(* Logix 5000 project; controller CLASE_1 Emulate 5570 rev 28.11; software revision 28.02 *)

TASK MainTask (continuous, watchdog 500 ms) : MainProgram
TASK TASK_A (periodic, rate 50 ms, priority 5, watchdog 150 ms) : Equipos_TK_100, Equipos_TK_200, Equipos_TK_300
TASK Task_B_100ms_Secuencias (periodic, rate 100 ms, priority 6, watchdog 300 ms) : SEC_Proceso_Chocolate_SFC
TASK Task_C_200ms (periodic, rate 200 ms, priority 7, watchdog 600 ms) : PID_Controllers

MODULES
   Local : Emulate 5570 (ICP 9, rev 28.11)
      Input_Digital_1 : 1756-IA16 (ICP 5, rev 3.1, Input RPI 20 ms)
      Output_Digital_2 : vendor 1 type 7 code 13 (ICP 6, rev 3.1, Output RPI 20 ms)
      input_analogica_1 : 1756-IF16 (ICP 7, rev 1.1, Input RPI 100 ms)
      Output_analogico_2 : 1756-OF8 (ICP 4, rev 1.1, Output RPI 12 ms)
END_MODULES

TYPE P_DescList :   // Code / Description List Entry
STRUCT
   Code : DINT;   // Code for which to look up Description
   Desc : STRING_40;   // Description for given Code
END_STRUCT
END_TYPE

TYPE STRING_12 :
STRUCT
   LEN : DINT;
   DATA : SINT[12];
END_STRUCT
END_TYPE

TYPE STRING_16 :
STRUCT
   LEN : DINT;
   DATA : SINT[16];
END_STRUCT
END_TYPE

TYPE STRING_20 :
STRUCT
   LEN : DINT;
   DATA : SINT[20];
END_STRUCT
END_TYPE

TYPE STRING_40 :
STRUCT
   LEN : DINT;
   DATA : SINT[40];
END_STRUCT
END_TYPE

TYPE STRING_8 :
STRUCT
   LEN : DINT;
   DATA : SINT[8];
END_STRUCT
END_TYPE

TYPE STRING_NavTag :   // Navigation Tag
STRUCT
   LEN : DINT;
   DATA : SINT[20];
END_STRUCT
END_TYPE

ADD_ON_INSTRUCTION P_AIn   (* revision 3.5 02 Release, vendor Rockwell Automation, ExecutePrescan, ExecuteEnableInFalse *)
// Analog Input
// Revision note:
// See V3.5-xx Release Notes for details. Added Cfg_UseChanSrcQ to make SrcQ use independent of Cfg_HasChanObj, which is for navigation only.
// Help:
// Copyright © Rockwell Automation, Inc.  All Rights Reserved.
// This Instruction monitors an Analog Input from a flow, level, pressure,
// temperature, or any other analog sensor, and provides:
// *  Scaling, from Input (Raw) to PV (Engineering) Units
// *  High-High, High, Low and Low-Low Status and Alarms, with Gate
// inputs and configurable on-delay, off-delay and gate delay times
// *  Monitoring of bad/uncertain PV status, floating point exceptions
// and out-of-range conditions, with PV Fail alarm
// *  Setting of a simulated input signal for process simulation
// *  Capturing of the lowest and highest PV excursion values
// *  Program and Operator Settings for Status Thresholds
// *  Configurable threshold deadbands and out of range limits
// *  Maintenance Commands to allow manual override of the input signal (Substitute PV)
// Modes are provided by a P_Mode AOI instance.
// Alarms are provided by P_Alarm AOI instances.
// Status gating provided by P_Gate AOI instances.
// Modes of operation: Operator, Program, Maintenance
VAR_INPUT
   Inp_PV : REAL; {visible}   // Input Signal (process variable) from Sensor
   Inp_PVSrcQ : SINT;   // Input Source and Quality (from Channel object, if available) (enum)
   Inp_PVBad : BOOL;   // 1=PV or I/O Comms Status Bad, 0=OK
   Inp_PVUncertain : BOOL;   // 1=PV Value Not Reliable, 0=OK
   Inp_Sim : BOOL;   // 1=Use simulated PV (Set_SimPV); 0=Use Input (Inp_PV)
   Inp_HiHiGate : ALIAS FOR HiHiGate.Inp_Gate;   // High-High Status Gate, 1=enabled
   Inp_HiGate : ALIAS FOR HiGate.Inp_Gate;   // High Status Gate, 1=enabled
   Inp_LoGate : ALIAS FOR LoGate.Inp_Gate;   // Low Status Gate, 1=enabled
   Inp_LoLoGate : ALIAS FOR LoLoGate.Inp_Gate;   // Low-Low Status Gate, 1=enabled
   Inp_FailGate : ALIAS FOR FailGate.Inp_Gate;   // Fail Status Gate, 1=enabled
   Inp_Reset : BOOL;   // 1=Reset all Alarms requiring reset
   Cfg_NoSubstPV : BOOL;   // 1=Disallow selection of Substitute PV
   Cfg_SetTrack : BOOL := 1;   // 1=PSets track OSets in Oper, OSets track PSets in Prog, 0=no tracking
   Cfg_HasChanObj : BOOL;   // 1=Tells HMI a Channel object (AIChan, etc.) is used for Inp_PV
   Cfg_UseChanSrcQ : BOOL;   // 1=Pass thru connected Channel's SrcQ value, 0=generate SrcQ
   Cfg_PCmdClear : ALIAS FOR Mode.Cfg_PCmdClear;
   Cfg_ProgDefault : ALIAS FOR Mode.Cfg_ProgDefault;
   Cfg_HasHiHiAlm : ALIAS FOR HiHi.Cfg_Exists;   // 1=High-High Alarm exists and will be checked
   Cfg_HasHiAlm : ALIAS FOR Hi.Cfg_Exists;   // 1=High Alarm exists and will be checked
   Cfg_HasLoAlm : ALIAS FOR Lo.Cfg_Exists;   // 1=Low Alarm exists and will be checked
   Cfg_HasLoLoAlm : ALIAS FOR LoLo.Cfg_Exists;   // 1=Low-Low Alarm exists and will be checked
   Cfg_HasFailAlm : ALIAS FOR Fail.Cfg_Exists;   // 1=Analog Input Failure Alarm exists and will be checked
   Cfg_HiHiResetReqd : ALIAS FOR HiHi.Cfg_ResetReqd;   // 1=Reset required to clear High-High Alarm
   Cfg_HiResetReqd : ALIAS FOR Hi.Cfg_ResetReqd;   // 1=Reset required to clear High Alarm
   Cfg_LoResetReqd : ALIAS FOR Lo.Cfg_ResetReqd;   // 1=Reset required to clear Low Alarm
   Cfg_LoLoResetReqd : ALIAS FOR LoLo.Cfg_ResetReqd;   // 1=Reset required to clear Low-Low Alarm
   Cfg_FailResetReqd : ALIAS FOR Fail.Cfg_ResetReqd;   // 1=Reset required to clear Analog InputFailure Alarm
   Cfg_HiHiAckReqd : ALIAS FOR HiHi.Cfg_AckReqd;   // 1=Acknowledge required for High-High Alarm
   Cfg_HiAckReqd : ALIAS FOR Hi.Cfg_AckReqd;   // 1=Acknowledge required for High Alarm
   Cfg_LoAckReqd : ALIAS FOR Lo.Cfg_AckReqd;   // 1=Acknlowledge required for Low Alarm
   Cfg_LoLoAckReqd : ALIAS FOR LoLo.Cfg_AckReqd;   // 1=Acknowledge required for Low-Low Alarm
   Cfg_FailAckReqd : ALIAS FOR Fail.Cfg_AckReqd;   // 1=Acknowledge required for Analog Input Failure Alarm
   Cfg_HiHiSeverity : ALIAS FOR HiHi.Cfg_Severity;   // High-High Alarm Severity: 1..250=Low, 251..500=Medium, 501..750=High, 751..1000=Urgent
   Cfg_HiSeverity : ALIAS FOR Hi.Cfg_Severity;   // High Alarm Severity: 1..250=Low, 251..500=Medium, 501..750=High, 751..1000=Urgent
   Cfg_LoSeverity : ALIAS FOR Lo.Cfg_Severity;   // Low Alarm Severity: 1..250=Low, 251..500=Medium, 501..750=High, 751..1000=Urgent
   Cfg_LoLoSeverity : ALIAS FOR LoLo.Cfg_Severity;   // Low-Low Alarm Severity: 1..250=Low, 251..500=Medium, 501..750=High, 751..1000=Urgent
   Cfg_FailSeverity : ALIAS FOR Fail.Cfg_Severity;   // Failure Alarm Severity: 1..250=Low, 251..500=Medium, 501..750=High, 751..1000=Urgent
   Cfg_InpRawMin : REAL;   // Input (unscaled) Minimum for Scaling
   Cfg_InpRawMax : REAL := 100.0;   // Input (unscaled) Maximum for Scaling
   Cfg_PVEUMin : REAL;   // PV (Output) Minimum for Scaling to EU
   Cfg_PVEUMax : REAL := 100.0;   // PV (Output) Maximum for Scaling to EU
   Cfg_FiltTC : REAL;   // PV Filter Time Constant (s), 0.0 = unfiltered
   Cfg_HiHiDB : REAL := 1.0;   // High-High Status Deadband (EU)
   Cfg_HiHiOnDly : ALIAS FOR HiHiGate.Cfg_OnDly;   // Minimum time above High-High Limit to raise Status (s)
   Cfg_HiHiOffDly : ALIAS FOR HiHiGate.Cfg_OffDly;   // Minimum time below High-High Limit (minus deadband) to clear Status (s)
   Cfg_HiHiGateDly : ALIAS FOR HiHiGate.Cfg_GateDly;   // High-High Status Gate Delay (s)
   Cfg_HiDB : REAL := 1.0;   // High Status Deadband (EU)
   Cfg_HiOnDly : ALIAS FOR HiGate.Cfg_OnDly;   // Minimum time above High Limit to raise Status (s)
   Cfg_HiOffDly : ALIAS FOR HiGate.Cfg_OffDly;   // Minimum time below High Limit (minus deadband) to clear Status (s)
   Cfg_HiGateDly : ALIAS FOR HiGate.Cfg_GateDly;   // High Status Gate Delay (s)
   Cfg_LoDB : REAL := 1.0;   // Low Status Deadband (EU)
   Cfg_LoOnDly : ALIAS FOR LoGate.Cfg_OnDly;   // Minimum time below Low Limit to raise Status (s)
   Cfg_LoOffDly : ALIAS FOR LoGate.Cfg_OffDly;   // Minimum time above Low Limit (plus deadband) to clear Status (s)
   Cfg_LoGateDly : ALIAS FOR LoGate.Cfg_GateDly;   // Low Status Gate Delay (s)
   Cfg_LoLoDB : REAL := 1.0;   // Low-Low Status Deadband (EU)
   Cfg_LoLoOnDly : ALIAS FOR LoLoGate.Cfg_OnDly;   // Minimum time below Low-Low Limit to raise Status (s)
   Cfg_LoLoOffDly : ALIAS FOR LoLoGate.Cfg_OffDly;   // Minimum time above Low-Low Limit (plus deadband) to clear Status (s)
   Cfg_LoLoGateDly : ALIAS FOR LoLoGate.Cfg_GateDly;   // Low-Low Status Gate Delay (s)
   Cfg_FailHiLim : REAL := 103.958336;   // Out-of-Range (fail) High Limit (EU)
   Cfg_FailLoLim : REAL := -2.0833333;   // Out-of-Range (fail) Low Limit (EU)
   Cfg_FailDB : REAL := 0.41666666;   // Out-of-Range (fail) High/Low Deadband (EU)
   Cfg_FailOnDly : ALIAS FOR FailGate.Cfg_OnDly;   // Minimum time Bad or Out of Range to raise Fail Status (s)
   Cfg_FailOffDly : ALIAS FOR FailGate.Cfg_OffDly;   // Minimum time OK or In Range to clear Fail Status (s)
   Cfg_FailGateDly : ALIAS FOR FailGate.Cfg_GateDly;   // Fail Status Gate Delay (s)
   PSet_Owner : DINT;   // Program Owner Request ID (non-zero) or Release (zero)
   PSet_HiHiLim : REAL := 1.5e+38;   // Program-Entered High-High Status Threshold (EU)
   PSet_HiLim : REAL := 1.5e+38;   // Program-Entered High Status Threshold (EU)
   PSet_LoLim : REAL := -1.5e+38;   // Program-Entered Low Status Threshold (EU)
   PSet_LoLoLim : REAL := -1.5e+38;   // Program-Entered Low-Low Status Threshold (EU)
   MSet_SubstPV : REAL;   // Maintenance-Entered Substitute PV (EU)
   OSet_HiHiLim : REAL := 1.5e+38;   // Operator-Entered High-High Status Threshold (EU)
   OSet_HiLim : REAL := 1.5e+38;   // Operator-Entered High Status Threshold (EU)
   OSet_LoLim : REAL := -1.5e+38;   // Operator-Entered Low Status Threshold (EU)
   OSet_LoLoLim : REAL := -1.5e+38;   // Operator-Entered Low-Low Status Threshold (EU)
   Set_SimPV : REAL;   // PV used in Simulation (Inp_Sim=1) (EU)
   PCmd_ClearCapt : BOOL;   // Program Command to Clear the captured min / max PV excursion values
   PCmd_Acq : ALIAS FOR Mode.PCmd_Acq;
   PCmd_Rel : ALIAS FOR Mode.PCmd_Rel;
   PCmd_Lock : ALIAS FOR Mode.PCmd_Lock;
   PCmd_Unlock : ALIAS FOR Mode.PCmd_Unlock;
   PCmd_Reset : BOOL;   // Program Command to Reset all Alarms requiring Reset
   PCmd_HiHiAck : ALIAS FOR HiHi.PCmd_Ack;   // Program Command to Acknowledge High-High Alarm
   PCmd_HiHiSuppress : ALIAS FOR HiHi.PCmd_Suppress;   // Program Command to Suppress High-High Alarm
   PCmd_HiHiUnsuppress : ALIAS FOR HiHi.PCmd_Unsuppress;   // Program Command to Unsuppress High-High Alarm
   PCmd_HiHiUnshelve : ALIAS FOR HiHi.PCmd_Unshelve;   // Program Command to Unshelve High-High Alarm
   PCmd_HiAck : ALIAS FOR Hi.PCmd_Ack;   // Program Command to Acknowledge High Alarm
   PCmd_HiSuppress : ALIAS FOR Hi.PCmd_Suppress;   // Program Command to Suppress High Alarm
   PCmd_HiUnsuppress : ALIAS FOR Hi.PCmd_Unsuppress;   // Program Command to Unsuppress High Alarm
   PCmd_HiUnshelve : ALIAS FOR Hi.PCmd_Unshelve;   // Program Command to Unshelve High Alarm
   PCmd_LoAck : ALIAS FOR Lo.PCmd_Ack;   // Program Command to Acknowledge Low Alarm
   PCmd_LoSuppress : ALIAS FOR Lo.PCmd_Suppress;   // Program Command to Suppress Low Alarm
   PCmd_LoUnsuppress : ALIAS FOR Lo.PCmd_Unsuppress;   // Program Command to Unsuppress Low Alarm
   PCmd_LoUnshelve : ALIAS FOR Lo.PCmd_Unshelve;   // Program Command to Unshelve Low Alarm
   PCmd_LoLoAck : ALIAS FOR LoLo.PCmd_Ack;   // Program Command to Acknowledge Low-Low Alarm
   PCmd_LoLoSuppress : ALIAS FOR LoLo.PCmd_Suppress;   // Program Command to Suppress Low-Low Alarm
   PCmd_LoLoUnsuppress : ALIAS FOR LoLo.PCmd_Unsuppress;   // Program Command to Unsuppress Low-Low Alarm
   PCmd_LoLoUnshelve : ALIAS FOR LoLo.PCmd_Unshelve;   // Program Command to Unshelve Low-Low Alarm
   PCmd_FailAck : ALIAS FOR Fail.PCmd_Ack;   // Program Command to Acknowldege Analog Input Failure Alarm
   PCmd_FailSuppress : ALIAS FOR Fail.PCmd_Suppress;   // Program Command to Suppress Analog Input Failure Alarm
   PCmd_FailUnsuppress : ALIAS FOR Fail.PCmd_Unsuppress;   // Program Command to Unsuppress Analog Input Failure Alarm
   PCmd_FailUnshelve : ALIAS FOR Fail.PCmd_Unshelve;   // Program Command to Unshelve Analog Input Failure Alarm
   MCmd_SubstPV : BOOL;   // Maintenance Command to use Substitute PV (override input)
   MCmd_InpPV : BOOL;   // Maintenance Command to use Input PV (normal)
   OCmd_ClearCapt : BOOL;   // Operator Command to Clear the captured min / max PV excursion values
   MCmd_Acq : ALIAS FOR Mode.MCmd_Acq;
   MCmd_Rel : ALIAS FOR Mode.MCmd_Rel;
   OCmd_AcqLock : ALIAS FOR Mode.OCmd_AcqLock;
   OCmd_Unlock : ALIAS FOR Mode.OCmd_UnlockRel;
   OCmd_Reset : BOOL;   // Operator Command to Reset all Alarms requiring Reset
   OCmd_ResetAckAll : BOOL;   // Operator Command to Reset and Acknowledge all Alarms
END_VAR
VAR_OUTPUT
   Val : REAL; {access Read Only, visible}   // Analog Value (after Substitute PV, if used)
   Val_InpPV : REAL; {access Read Only, visible}   // Analog Input Value (actual, before Substitute PV selection)
   Val_PVMinCapt : REAL := 1.5e+38; {access Read Only}   // Captured PV Minimum (excursion) since last cleared
   Val_PVMaxCapt : REAL := -1.5e+38; {access Read Only}   // Captured PV Maximum (excursion) since last cleared
   Val_PVEUMin : REAL; {access Read Only}   // Minimum of scaled range = MIN (Cfg_PVEUMin, Cfg_PVEUMax)
   Val_PVEUMax : REAL := 100.0; {access Read Only}   // Maximum of scaled range = MAX (Cfg_PVEUMin, Cfg_PVEUMax)
   SrcQ_IO : SINT; {access Read Only}   // Source and Quality of primary I/O (enumeration)
   SrcQ : SINT; {access Read Only}   // Source and Quality of primary Val/Sts (enumeration)
   Val_Fault : SINT; {access Read Only}   // Device Fault Status 0=none, 20=Lo, 21=Hi, 24=LoLo, 25=HiHi, 32=Fail, 34=CfgErr
   Val_Mode : ALIAS FOR Mode.Val; {access Read Only}
   Val_Owner : DINT; {access Read Only}   // Current Object Owner ID (0=not owned)
   Val_Notify : SINT; {access Read Only}   // Current Alarm Level and Acknowledgement (enumeration)
   Val_HiHiLim : REAL := 1.5e+38; {access Read Only, visible}   // Current High-High Status Threshold
   Val_HiLim : REAL := 1.5e+38; {access Read Only, visible}   // Current High Status Threshold
   Val_LoLim : REAL := -1.5e+38; {access Read Only, visible}   // Current Low Status Threshold
   Val_LoLoLim : REAL := -1.5e+38; {access Read Only, visible}   // Current Low-Low Status Threshold
   Sts_SubstPV : BOOL; {access Read Only}   // 1=Using Substitute PV (Input being overridden)
   Sts_InpPV : BOOL := 1; {access Read Only}   // 1=Using Input PV (normal)
   Sts_PVBad : BOOL; {access Read Only}   // 1=PV Bad quality or Out of Range
   Sts_PVUncertain : BOOL; {access Read Only}   // 1=PV Value is Uncertain (quality)
   Sts_MaintByp : BOOL; {access Read Only}   // 1=A Maintenance Bypass is Active, display icon
   Sts_AlmInh : BOOL; {access Read Only}   // 1=An Alarm is Shelved, Disabled or Suppressed: display icon
   Sts_Err : BOOL; {access Read Only, visible}   // 1=Error in Config (see detail Err_ bits for reason), display icon
   Err_Raw : BOOL; {access Read Only}   // 1=Error in Config: Raw Input Scaling Min = Max
   Err_EU : BOOL; {access Read Only}   // 1=Error in Config: Scaled EU Min = Max
   Err_Timer : BOOL; {access Read Only}   // 1=Error in Config: On Delay, Off Delay, Gate Delay Time Invalid (use 0 to 2147483 s)
   Err_Filt : BOOL; {access Read Only}   // 1=Error in Config: PV filter params (RateTime, TC)
   Err_DB : BOOL; {access Read Only}   // 1=Error in Config: a Status Deadband is < 0.0
   Err_Alarm : BOOL; {access Read Only}   // 1=Error in Config: Alarm Min On Time, Shelf Time, Severity
   Sts_Maint : ALIAS FOR Mode.Sts_Maint; {access Read Only}
   Sts_Prog : ALIAS FOR Mode.Sts_Prog; {access Read Only}
   Sts_Oper : ALIAS FOR Mode.Sts_Oper; {access Read Only}
   Sts_ProgOperLock : ALIAS FOR Mode.Sts_ProgOperLock; {access Read Only}
   Sts_NoMode : ALIAS FOR Mode.Sts_NoMode; {access Read Only}
   Sts_MAcqRcvd : ALIAS FOR Mode.Sts_MAcqRcvd; {access Read Only}
   Sts_HiHiCmp : ALIAS FOR HiHiGate.Inp;   // PV High-High comparison result 1=High-High
   Sts_HiHiGate : ALIAS FOR HiHiGate.Sts_Gate; {access Read Only}   // PV High-High Gate Delay Status, 1=done
   Sts_HiHi : ALIAS FOR HiHi.Inp;   // 1=Analog Input is above High-High limit
   Alm_HiHi : ALIAS FOR HiHi.Alm;   // 1=Analog Input is in High-High Alarm
   Ack_HiHi : ALIAS FOR HiHi.Ack;   // 1=High-High Alarm has been acknowledged
   Sts_HiHiDisabled : ALIAS FOR HiHi.Disabled;   // 1=High-High Alarm has been Disabled by Maintenancy
   Sts_HiHiSuppressed : ALIAS FOR HiHi.Suppressed;   // 1=High-High Alarm has been Suppressed by Program
   Sts_HiHiShelved : ALIAS FOR HiHi.Shelved;   // 1=High-High Alarm has been Shelved by Operator
   Sts_HiCmp : ALIAS FOR HiGate.Inp;   // PV High comparison result 1=High
   Sts_HiGate : ALIAS FOR HiGate.Sts_Gate; {access Read Only}   // PV High Gate Delay Status, 1=done
   Sts_Hi : ALIAS FOR Hi.Inp;   // 1=Analog Input is above High limit
   Alm_Hi : ALIAS FOR Hi.Alm;   // 1=Analog Input is in High Alarm
   Ack_Hi : ALIAS FOR Hi.Ack;   // 1=High Alarm has been acknowledged
   Sts_HiDisabled : ALIAS FOR Hi.Disabled;   // 1=High Alarm has been Disabled by Maintenance
   Sts_HiSuppressed : ALIAS FOR Hi.Suppressed;   // 1=High Alarm has been Suppressed by Program
   Sts_HiShelved : ALIAS FOR Hi.Shelved;   // 1=High Alarm has been Shelved by Operator
   Sts_LoCmp : ALIAS FOR LoGate.Inp;   // PV Low comparison result 1=Low
   Sts_LoGate : ALIAS FOR LoGate.Sts_Gate; {access Read Only}   // PV Low Gate Delay Status, 1=done
   Sts_Lo : ALIAS FOR Lo.Inp;   // 1=Analog Input is below Low limit
   Alm_Lo : ALIAS FOR Lo.Alm;   // 1=Analog Input is in Low Alarm
   Ack_Lo : ALIAS FOR Lo.Ack;   // 1=Low Alarm has been acknowledged
   Sts_LoDisabled : ALIAS FOR Lo.Disabled;   // 1=Low Alarm has been Disabled by Maintenance
   Sts_LoSuppressed : ALIAS FOR Lo.Suppressed;   // 1=Low Alarm has been Suppressed by Program
   Sts_LoShelved : ALIAS FOR Lo.Shelved;   // 1=Low Alarm has been Shelved by Operator
   Sts_LoLoCmp : ALIAS FOR LoLoGate.Inp;   // PV Low-Low comparison result 1=Low-Low
   Sts_LoLoGate : ALIAS FOR LoLoGate.Sts_Gate; {access Read Only}   // PV Low-Low Gate Delay Status, 1=done
   Sts_LoLo : ALIAS FOR LoLo.Inp;   // 1=Analog Input is below Low-Low limit
   Alm_LoLo : ALIAS FOR LoLo.Alm;   // 1=Analog Input is in Low-Low Alarm
   Ack_LoLo : ALIAS FOR LoLo.Ack;   // 1=Low-Low Alarm has been acknowledged
   Sts_LoLoDisabled : ALIAS FOR LoLo.Disabled;   // 1=Low-Low Alarm has been Disabled by Maintenance
   Sts_LoLoSuppressed : ALIAS FOR LoLo.Suppressed;   // 1=Low-Low Alarm has been Suppressed by Program
   Sts_LoLoShelved : ALIAS FOR LoLo.Shelved;   // 1=Low-Low Alarm has been Shelved by Operator
   Sts_FailCmp : ALIAS FOR FailGate.Inp;   // PV Fail comparison result 1=Out of Range
   Sts_FailGate : ALIAS FOR FailGate.Sts_Gate; {access Read Only}   // PV Fail Gate Delay Status, 1=done
   Sts_Fail : ALIAS FOR Fail.Inp;   // 1=Analog Input is Out of Range or PV Bad
   Alm_Fail : ALIAS FOR Fail.Alm;   // 1=Analog Input Failure Alarm (PV Bad or Out of Range)
   Ack_Fail : ALIAS FOR Fail.Ack;   // 1=Analog Input Failure Alarm has been acknowledged
   Sts_FailDisabled : ALIAS FOR Fail.Disabled;   // 1=Analog input Failure Alarm has been Disabled by Maintenance
   Sts_FailSuppressed : ALIAS FOR Fail.Suppressed;   // 1=Analog Input Failure Alarm has been Suppressed by Program
   Sts_FailShelved : ALIAS FOR Fail.Shelved;   // 1=Analog Input Failure Alarm has been Shelved by Operator
   Rdy_SubstPV : BOOL; {access Read Only}   // 1=Ready for MCmd_SubstPV
   Rdy_InpPV : BOOL; {access Read Only}   // 1=Ready for MCmd_InpPV
   Rdy_Reset : BOOL; {access Read Only}   // 1=At least one Alarm requires Reset
   Rdy_ResetAckAll : BOOL; {access Read Only}   // 1=At least one Alarm requires Reset or Acknowledgement
   Rdy_OSet : BOOL; {access Read Only}   // 1=Ready to receive OSets (enables data entry fields)
   P_AIn : BOOL;   // Unique Parameter Name for auto - discovery
END_VAR
VAR
   LoLo : P_Alarm := (Cfg_AckReqd := 1, Cfg_AllowShelve := 1, Cfg_AllowDisable := 1, Cfg_PCmdClear := 1, Cfg_Severity := 750, Cfg_AlmMinOnT := 5, PCfg_AllowExist := 1, Ack := 1);   // Low-Low Alarm
   Lo : P_Alarm := (Cfg_AckReqd := 1, Cfg_AllowShelve := 1, Cfg_AllowDisable := 1, Cfg_PCmdClear := 1, Cfg_Severity := 500, Cfg_AlmMinOnT := 5, PCfg_AllowExist := 1, Ack := 1);   // Low Alarm
   Hi : P_Alarm := (Cfg_AckReqd := 1, Cfg_AllowShelve := 1, Cfg_AllowDisable := 1, Cfg_PCmdClear := 1, Cfg_Severity := 500, Cfg_AlmMinOnT := 5, PCfg_AllowExist := 1, Ack := 1);   // High Alarm
   HiHi : P_Alarm := (Cfg_AckReqd := 1, Cfg_AllowShelve := 1, Cfg_AllowDisable := 1, Cfg_PCmdClear := 1, Cfg_Severity := 750, Cfg_AlmMinOnT := 5, PCfg_AllowExist := 1, Ack := 1);   // High-High Alarm
   Mode : P_Mode := (Cfg_PCmdClear := 1, Cfg_OvrdOverLock := 1, Sts_Oper := 1, Rdy_MRel := 1, Rdy_OAcq := 1);   // Analog Input Mode Selection
   Cfg_EU : STRING_8 := '%';   // Engineering Units for display on HMI
   Cfg_Tag : STRING_20 := 'P_AIn';   // Tagname for display on HMI
   Cfg_Label : STRING_20 := 'Analog Input';   // Label for graphic symbol displayed on HMI
   Cfg_Desc : STRING_40 := 'Analog Input';   // Description for display on HMI
   Fail : P_Alarm := (Cfg_AckReqd := 1, Cfg_AllowShelve := 1, Cfg_AllowDisable := 1, Cfg_PCmdClear := 1, Cfg_Severity := 1000, Cfg_AlmMinOnT := 5, PCfg_AllowExist := 1, Ack := 1);   // Analog Input Failure Alarm (bad quality or out of range)
   Wrk_Notify : SINT; {access None}   // Buffer for building Val_Notify
   Inf_Tab : SINT;   // Tab to display (FTView ME)
   Wrk_Fault : SINT; {access None}   // Buffer for building Val_Fault
   Wrk_SrcQ : SINT; {access None}   // Register for building Source / Quality enumeration
   Wrk_SubstPV : BOOL; {access None}   // Internal flag: Using Substitute PV
   Wrk_UnfiltPV : REAL; {access None}   // Unfiltered PV, input to 1st order filter
   Wrk_Alpha : REAL; {access None}   // Filter multiplier = (1 / (1+TC/dT) )
   Wrk_ScanT : TIMER := (PRE := 2147483647); {access None}   // Scan Timer (milliseconds, always runs)
   Wrk_ScanTime : REAL; {access None}   // Time since this instance was last scanned
   Wrk_FiltPV : REAL; {access None}   // Filtered PV
   Wrk_ValidONS : BOOL; {access None}   // Selected PV goes from Infinite or Not a Number to VALID
   Wrk_SelPVDINT : DINT; {access None}   // Selected PV check for Infinite or Non A Number
   Wrk_SelPVInfNaN : BOOL; {access None}   // Selected PV (Input or Substitute) is Infinite or NaN
   Inf_Type : STRING_16 := 'P_AIn'; {access Read Only}   // Must contain AOI name, used for HMI and Information S/W
   Wrk_Fail : BOOL; {access None}   // Internal flag: Fail Status
   Wrk_LoLo : BOOL; {access None}   // Internal flag: Low-Low Status
   Wrk_Lo : BOOL; {access None}   // Internal flag: Low Status
   Wrk_Hi : BOOL; {access None}   // Internal flag: High Status
   Wrk_HiHi : BOOL; {access None}   // Internal flag: High-High Status
   FailGate : P_Gate := (Inp_Gate := 1);   // Fail Alarm Gate / Delay Block
   LoLoGate : P_Gate := (Inp_Gate := 1);   // Low-Low Alarm Gate / Delay Block
   LoGate : P_Gate := (Inp_Gate := 1);   // Low Alarm Gate / Delay Block
   HiHiGate : P_Gate := (Inp_Gate := 1);   // High-High Alarm Gate / Delay Block
   HiGate : P_Gate := (Inp_Gate := 1);   // High Alarm Gate / Delay Block
   Wrk_InpInfNaN : BOOL; {access None}   // Input is Infinite or Not a Number
   Wrk_InpDINT : DINT; {access None}   // Input REAL bit pattern as a DINT (check for Inf/NaN)
   Inf_Lib : STRING_12 := 'RA-BAS'; {access Read Only}   // Display Library for Faceplate call-up
   Wrk_InpFail : BOOL; {access None}   // Input Fail: out of range
END_VAR

ROUTINE EnableInFalse   (* ladder *)
// Off-Scan: no Val update or alarm checking.  PV Bad Quality ("stale") is asserted.
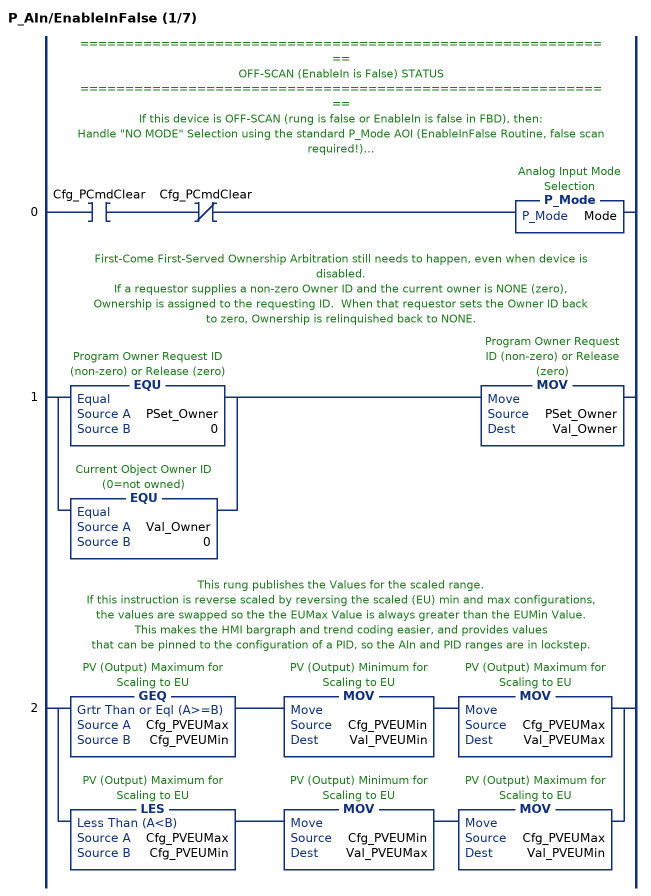
   // ============================================================
   // OFF-SCAN (EnableIn is False) STATUS
   // ============================================================
   // If this device is OFF-SCAN (rung is false or EnableIn is false in FBD), then:
   // Handle "NO MODE" Selection using the standard P_Mode AOI (EnableInFalse Routine, false scan required!).
   // NOTE:  IN ORDER TO AVOID USING AN "AFI" (which will generate a routine verify warning),
   // THIS RUNG USES AN XIC of Cfg_PCmdClear, followed by an XIO of the SAME BIT
   // to ensure P_Mode is SCANNED FALSE ("NO MODE").
   // THIS IS NOT DEAD CODE AND MUST APPEAR EXACTLY AS SHOWN FOR PROPER OPERATION!
   0: XIC(Cfg_PCmdClear)XIO(Cfg_PCmdClear)P_Mode(Mode);
   // First-Come First-Served Ownership Arbitration still needs to happen, even when device is disabled.
   // If a requestor supplies a non-zero Owner ID and the current owner is NONE (zero),
   // Ownership is assigned to the requesting ID.  When that requestor sets the Owner ID back
   // to zero, Ownership is relinquished back to NONE.
   1: [EQU(PSet_Owner,0) ,EQU(Val_Owner,0) ]MOV(PSet_Owner,Val_Owner);
   // This rung publishes the Values for the scaled range.
   // If this instruction is reverse scaled by reversing the scaled (EU) min and max configurations,
   // the values are swapped so the the EUMax Value is always greater than the EUMin Value.
   // This makes the HMI bargraph and trend coding easier, and provides values
   // that can be pinned to the configuration of a PID, so the AIn and PID ranges are in lockstep.
   2: [GEQ(Cfg_PVEUMax,Cfg_PVEUMin) MOV(Cfg_PVEUMin,Val_PVEUMin) MOV(Cfg_PVEUMax,Val_PVEUMax) ,LES(Cfg_PVEUMax,Cfg_PVEUMin) MOV(Cfg_PVEUMin,Val_PVEUMax) MOV(Cfg_PVEUMax,Val_PVEUMin) ];
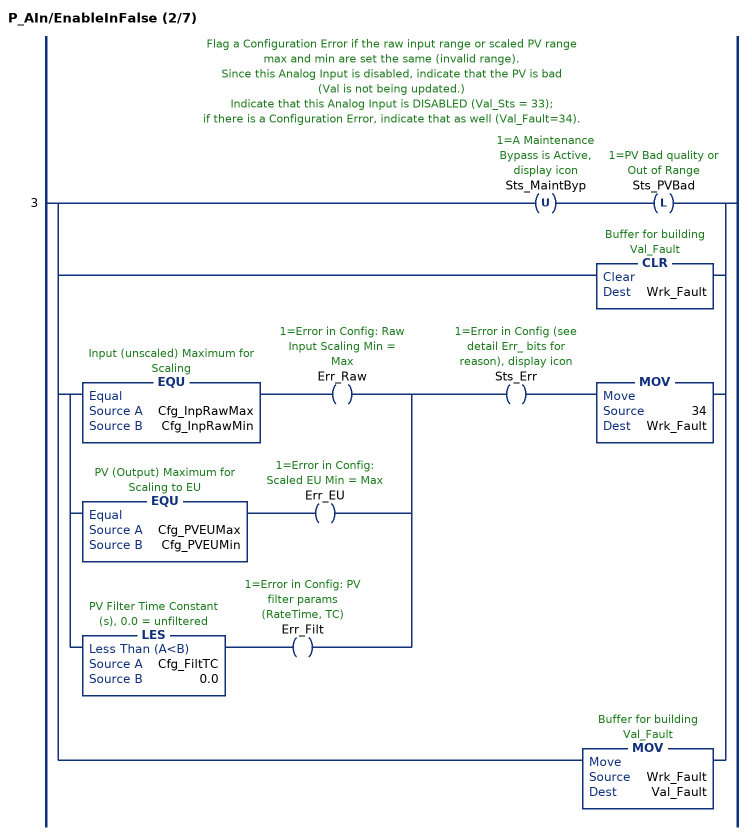
   // Flag a Configuration Error if the raw input range or scaled PV range
   // max and min are set the same (invalid range).
   // Since this Analog Input is disabled, indicate that the PV is bad
   // (Val is not being updated.)
   // Indicate that this Analog Input is DISABLED (Val_Sts = 33);
   // if there is a Configuration Error, indicate that as well (Val_Fault=34).
   3: [OTU(Sts_MaintByp) OTL(Sts_PVBad) ,CLR(Wrk_Fault) ,[EQU(Cfg_InpRawMax,Cfg_InpRawMin) OTE(Err_Raw) ,EQU(Cfg_PVEUMax,Cfg_PVEUMin) OTE(Err_EU) ,LES(Cfg_FiltTC,0.0) OTE(Err_Filt) ] OTE(Sts_Err) MOV(34,Wrk_Fault) ,MOV(Wrk_Fault,Val_Fault) ];
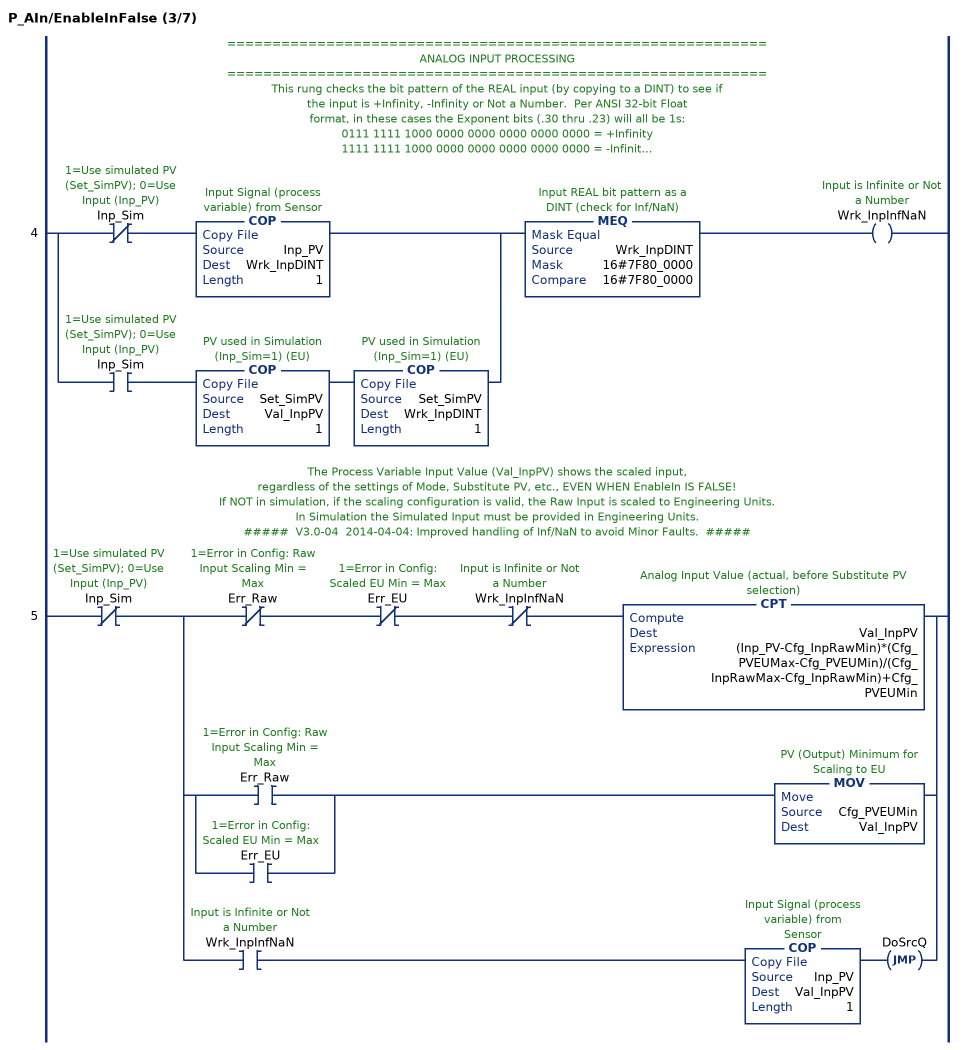
   // ============================================================
   // ANALOG INPUT PROCESSING
   // ============================================================
   // This rung checks the bit pattern of the REAL input (by copying to a DINT) to see if
   // the input is +Infinity, -Infinity or Not a Number.  Per ANSI 32-bit Float
   // format, in these cases the Exponent bits (.30 thru .23) will all be 1s:
   // 0111 1111 1000 0000 0000 0000 0000 0000 = +Infinity
   // 1111 1111 1000 0000 0000 0000 0000 0000 = -Infinity
   // x111 1111 1xxx xxxx xxxx xxxx xxxx xxxx = Not a Number
   // #####  V3.0-04  2014-04-04: Improved handling of Inf/NaN to avoid Minor Faults.  #####
   4: [XIO(Inp_Sim) COP(Inp_PV,Wrk_InpDINT,1) ,XIC(Inp_Sim) COP(Set_SimPV,Val_InpPV,1) COP(Set_SimPV,Wrk_InpDINT,1) ]MEQ(Wrk_InpDINT,16#7F80_0000,16#7F80_0000)OTE(Wrk_InpInfNaN);
   // The Process Variable Input Value (Val_InpPV) shows the scaled input,
   // regardless of the settings of Mode, Substitute PV, etc., EVEN WHEN EnableIn IS FALSE!
   // If NOT in simulation, if the scaling configuration is valid, the Raw Input is scaled to Engineering Units.
   // In Simulation the Simulated Input must be provided in Engineering Units.
   // #####  V3.0-04  2014-04-04: Improved handling of Inf/NaN to avoid Minor Faults.  #####
   5: XIO(Inp_Sim)[XIO(Err_Raw) XIO(Err_EU) XIO(Wrk_InpInfNaN) CPT(Val_InpPV,(Inp_PV-Cfg_InpRawMin)*(Cfg_PVEUMax-Cfg_PVEUMin)/(Cfg_InpRawMax-Cfg_InpRawMin)+Cfg_PVEUMin) ,[XIC(Err_Raw) ,XIC(Err_EU) ] MOV(Cfg_PVEUMin,Val_InpPV) ,XIC(Wrk_InpInfNaN) COP(Inp_PV,Val_InpPV,1) JMP(DoSrcQ) ];
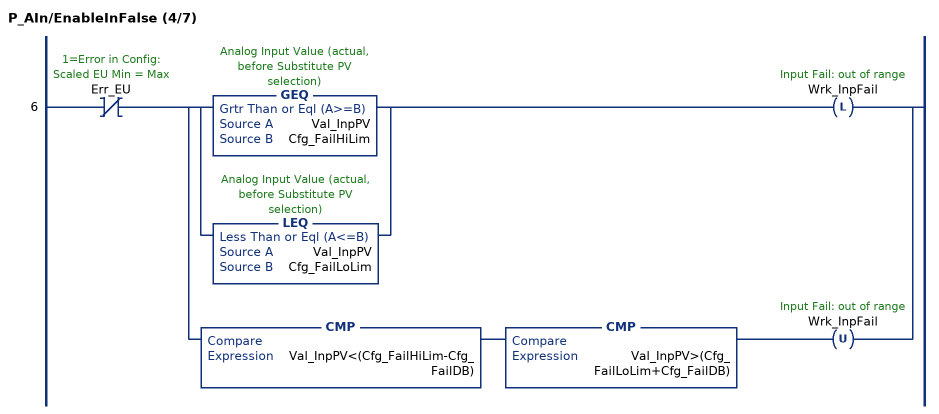
   6: XIO(Err_EU)[[GEQ(Val_InpPV,Cfg_FailHiLim) ,LEQ(Val_InpPV,Cfg_FailLoLim) ] OTL(Wrk_InpFail) ,CMP(Val_InpPV<(Cfg_FailHiLim-Cfg_FailDB)) CMP(Val_InpPV>(Cfg_FailLoLim+Cfg_FailDB)) OTU(Wrk_InpFail) ];
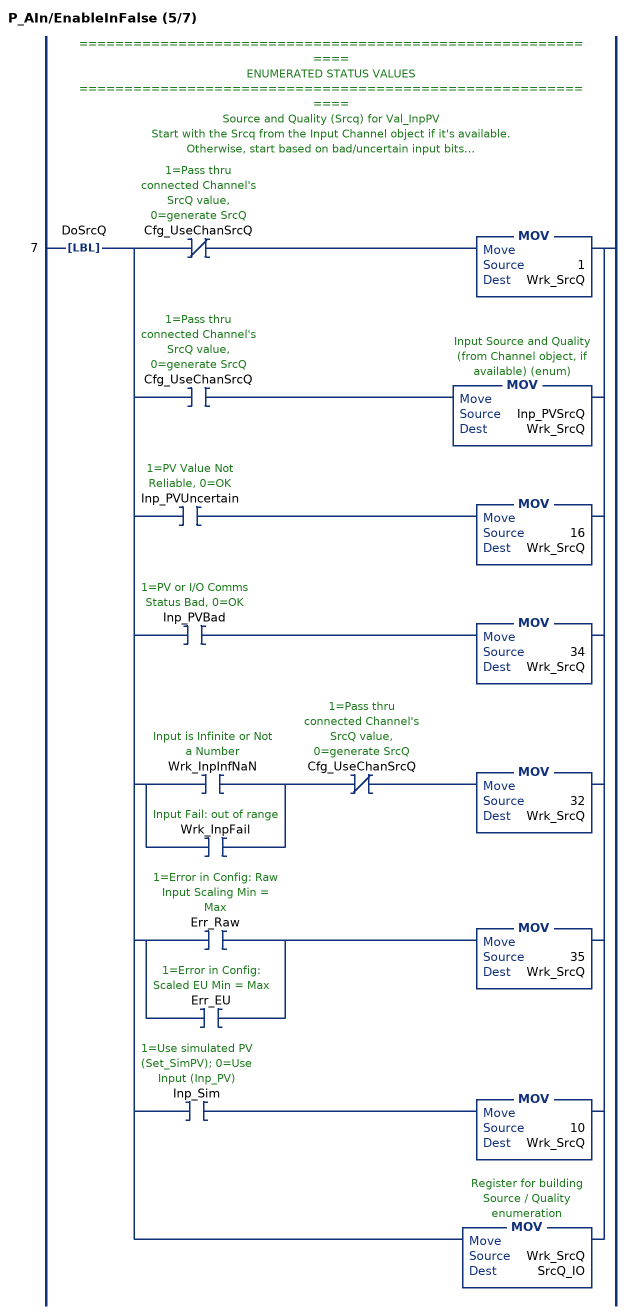
   // ============================================================
   // ENUMERATED STATUS VALUES
   // ============================================================
   // Source and Quality (Srcq) for Val_InpPV
   // Start with the Srcq from the Input Channel object if it's available.
   // Otherwise, start based on bad/uncertain input bits.
   // 0 = Good: live, confirmed good;   1 = Good: live, assumed good;
   // 8 = Test: Simulated;   9 = Test: Loopback;
   // 10 = Test: Manually Entered;   16 = Uncertain: Live, off-spec;
   // 17 = Uncertain, Substituted at Device / Bus;   18 = Uncertain, Substituted at AOI;
   // 19 = Uncertain, using last known good;    20 = Uncertain, using replacement value;
   // 32 = Bad, Signal Failure;   33 = Bad, Channel Fault;
   // 34 = Bad, Module / Comms Fault;   35 = Bad, Invalid Configuration
   // #####  V3.1-00  2014-06-30:  Added rung for Source/Quality enumerations.  #####
   // #####  V3.5-02  2016-03-28:  Modified to add Cfg_UseChanSrcQ.  #####
   7: LBL(DoSrcQ)[XIO(Cfg_UseChanSrcQ) MOV(1,Wrk_SrcQ) ,XIC(Cfg_UseChanSrcQ) MOV(Inp_PVSrcQ,Wrk_SrcQ) ,XIC(Inp_PVUncertain) MOV(16,Wrk_SrcQ) ,XIC(Inp_PVBad) MOV(34,Wrk_SrcQ) ,[XIC(Wrk_InpInfNaN) ,XIC(Wrk_InpFail) ] XIO(Cfg_UseChanSrcQ) MOV(32,Wrk_SrcQ) ,[XIC(Err_Raw) ,XIC(Err_EU) ] MOV(35,Wrk_SrcQ) ,XIC(Inp_Sim) MOV(10,Wrk_SrcQ) ,MOV(Wrk_SrcQ,SrcQ_IO) ];
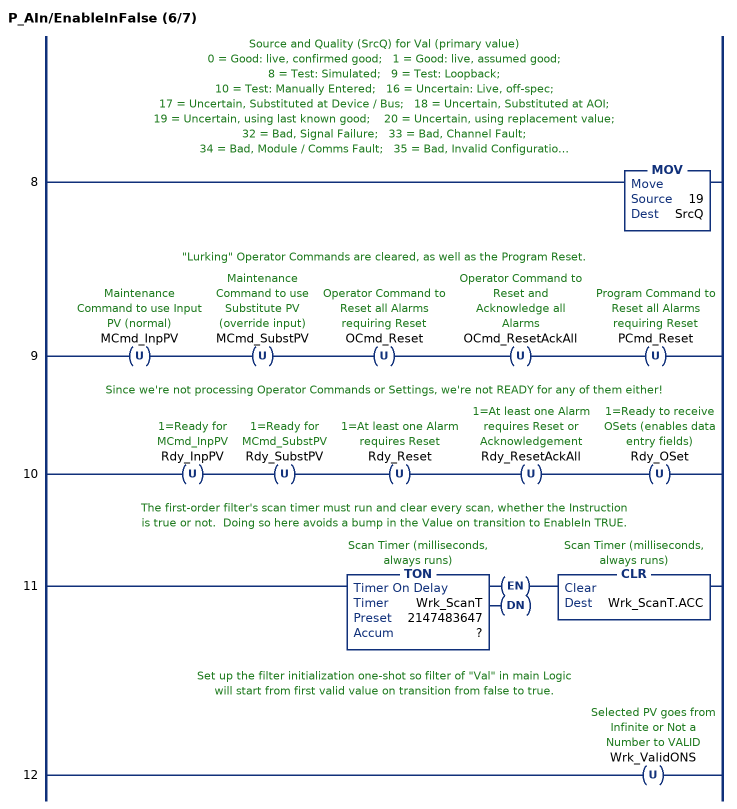
   // Source and Quality (SrcQ) for Val (primary value)
   // 0 = Good: live, confirmed good;   1 = Good: live, assumed good;
   // 8 = Test: Simulated;   9 = Test: Loopback;
   // 10 = Test: Manually Entered;   16 = Uncertain: Live, off-spec;
   // 17 = Uncertain, Substituted at Device / Bus;   18 = Uncertain, Substituted at AOI;
   // 19 = Uncertain, using last known good;    20 = Uncertain, using replacement value;
   // 32 = Bad, Signal Failure;   33 = Bad, Channel Fault;
   // 34 = Bad, Module / Comms Fault;   35 = Bad, Invalid Configuration
   // #####  V3.1-00  2014-06-30:  Added rung for Source/Quality enumerations.  #####
   8: MOV(19,SrcQ);
   // "Lurking" Operator Commands are cleared, as well as the Program Reset.
   9: OTU(MCmd_InpPV)OTU(MCmd_SubstPV)OTU(OCmd_Reset)OTU(OCmd_ResetAckAll)OTU(PCmd_Reset);
   // Since we're not processing Operator Commands or Settings, we're not READY for any of them either!
   10: OTU(Rdy_InpPV)OTU(Rdy_SubstPV)OTU(Rdy_Reset)OTU(Rdy_ResetAckAll)OTU(Rdy_OSet);
   // The first-order filter's scan timer must run and clear every scan, whether the Instruction
   // is true or not.  Doing so here avoids a bump in the Value on transition to EnableIn TRUE.
   11: TON(Wrk_ScanT,?,?)CLR(Wrk_ScanT.ACC);
   // Set up the filter initialization one-shot so filter of "Val" in main Logic
   // will start from first valid value on transition from false to true.
   12: OTU(Wrk_ValidONS);
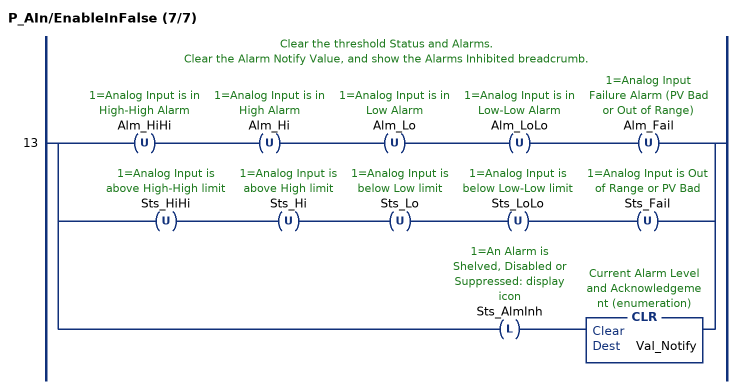
   // Clear the threshold Status and Alarms.
   // Clear the Alarm Notify Value, and show the Alarms Inhibited breadcrumb.
   13: [OTU(Alm_HiHi) OTU(Alm_Hi) OTU(Alm_Lo) OTU(Alm_LoLo) OTU(Alm_Fail) ,OTU(Sts_HiHi) OTU(Sts_Hi) OTU(Sts_Lo) OTU(Sts_LoLo) OTU(Sts_Fail) ,OTL(Sts_AlmInh) CLR(Val_Notify) ];
END_ROUTINE

ROUTINE Logic   (* ladder *)
// Normal Scan - PV is scaled and alarms are generated
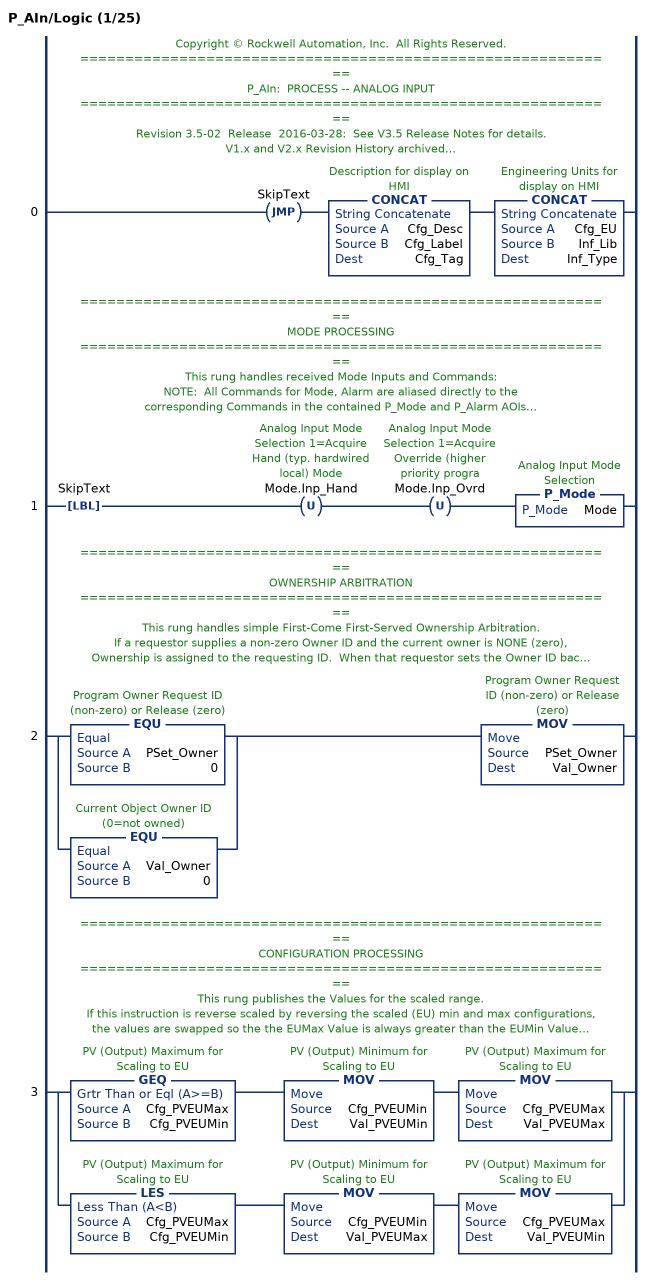
   // Copyright © Rockwell Automation, Inc.  All Rights Reserved.
   // ============================================================
   // P_AIn:  PROCESS -- ANALOG INPUT
   // ============================================================
   // Revision 3.5-02  Release  2016-03-28:  See V3.5 Release Notes for details.
   // V1.x and V2.x Revision History archived.
   // V3.0-00  2013-06-30:  Uses P_Gate, P_Alarm, P_Mode V3.0.
   // Added Inf_Lib, navigation to Channel obj.
   // V3.0-01  2013-07-30:  Modified Parameter descriptions only.
   // V3.0-02  2013-09-03:  Modified Parameter descriptions only.
   // V3.0-03  2013-10-30:  Corrected Parameter descriptions and default
   // configuration values for alarms only.
   // V3.0-04  2014-04-04:   Improved handling of Inf/NaN to avoid Minor Faults.
   // V3.1-00  2014-07-08:  Modified to use P_Alarm, P_Mode V3.1, add SrcQ enums.
   // Modified to consistently use alias tag names.
   // V3.1-01  2014-09-03:  Inp_PVSrcQ pulled into all bad/uncertain logic.
   // Using P_Alarm, P_Gate, P_Mode V3.1-01.
   // V3.1-02  2014-09-30:  Unchanged, but using P_Alarm V3.1-02.
   // V3.1-05  2016-01-22:  Added check of SrcQ >= 32 for Val_Fault.
   // Changed default values of min, max capture. Modified to
   // handle on-delay near status thresholds properly.
   // V3.5-01  2016-01-29:  Unchanged, using P_Alarm, P_Gate V3.5-01.
   // V3.5-02  2016-03-28:  Added Cfg_UseChanSrcQ to make SrcQ use
   // independent of Cfg_HasChanObj, which is for navigation only.
   // ============================================================
   // This Instruction monitors an Analog Input from a flow, level, pressure,
   // temperature, or any other analog sensor, and provides:
   // *  Scaling, from Input (Raw) to PV (Engineering) Units
   // *  High-High, High, Low and Low-Low Status and Alarms, with Gate
   // inputs and configurable on-delay, off-delay and gate delay times
   // *  Monitoring of bad/uncertain PV status, floating point exceptions
   // and out-of-range conditions, with PV Fail alarm
   // *  Setting of a simulated input signal for process simulation
   // *  Capturing of the lowest and highest PV excursion values
   // *  Program and Operator Settings for Status Thresholds
   // *  Configurable threshold deadbands and out of range limits
   // *  Maintenance Commands to allow manual override of the input signal (Substitute PV)
   // Modes are provided by a P_Mode AOI instance.
   // Alarms are provided by P_Alarm AOI instances.
   // Status gating provided by P_Gate AOI instances.
   // Modes of operation: Operator, Program, Maintenance
   // ============================================================
   // SHOW LOCAL STRINGS
   // ============================================================
   // The STRINGs containing the text associated with each instance of this
   // instruction cannot be Input or Output Parameters, because STRINGs are not
   //  'atomic' types. (Inputs and Outputs must be SINT, INT, DINT, REAL, or BOOL.)
   // In order to make it easier to find and configure these STRINGs, this rung
   // was added.  THE JMP (and the LBL on the following rung)
   // MUST NOT BE REMOVED!!!
   // To view the STRINGs, go to the instruction instance (in LD or FBD), RIGHT-click
   // to bring up the context menu and select "Open Instruction Logic".
   // This rung will appear with the STRING values for the selected instance.
   // You may double-click the STRING values here to modify them as well.
   // #####  V3.0-00  2013-06-30:  Added Inf_Lib  #####
   0: JMP(SkipText)CONCAT(Cfg_Desc,Cfg_Label,Cfg_Tag)CONCAT(Cfg_EU,Inf_Lib,Inf_Type);
   // ============================================================
   // MODE PROCESSING
   // ============================================================
   // This rung handles received Mode Inputs and Commands:
   // NOTE:  All Commands for Mode, Alarm are aliased directly to the
   // corresponding Commands in the contained P_Mode and P_Alarm AOIs.
   // This object does NOT have the following Modes:
   // Hand
   // Override
   1: LBL(SkipText)OTU(Mode.Inp_Hand)OTU(Mode.Inp_Ovrd)P_Mode(Mode);
   // ============================================================
   // OWNERSHIP ARBITRATION
   // ============================================================
   // This rung handles simple First-Come First-Served Ownership Arbitration.
   // If a requestor supplies a non-zero Owner ID and the current owner is NONE (zero),
   // Ownership is assigned to the requesting ID.  When that requestor sets the Owner ID back
   // to zero, Ownership is relinquished back to NONE.
   2: [EQU(PSet_Owner,0) ,EQU(Val_Owner,0) ]MOV(PSet_Owner,Val_Owner);
   // ============================================================
   // CONFIGURATION PROCESSING
   // ============================================================
   // This rung publishes the Values for the scaled range.
   // If this instruction is reverse scaled by reversing the scaled (EU) min and max configurations,
   // the values are swapped so the the EUMax Value is always greater than the EUMin Value.
   // This makes the HMI bargraph and trend coding easier, and provides values
   // that can be pinned to the configuration of a PID, so the AIn and PID ranges are in lockstep.
   3: [GEQ(Cfg_PVEUMax,Cfg_PVEUMin) MOV(Cfg_PVEUMin,Val_PVEUMin) MOV(Cfg_PVEUMax,Val_PVEUMax) ,LES(Cfg_PVEUMax,Cfg_PVEUMin) MOV(Cfg_PVEUMin,Val_PVEUMax) MOV(Cfg_PVEUMax,Val_PVEUMin) ];
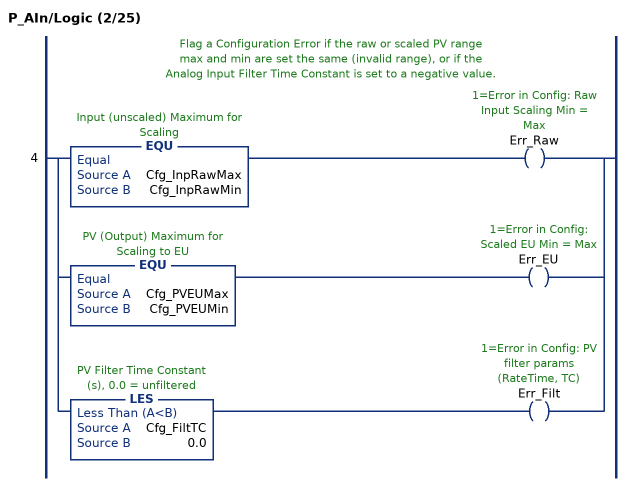
   // Flag a Configuration Error if the raw or scaled PV range
   // max and min are set the same (invalid range), or if the
   // Analog Input Filter Time Constant is set to a negative value.
   4: [EQU(Cfg_InpRawMax,Cfg_InpRawMin) OTE(Err_Raw) ,EQU(Cfg_PVEUMax,Cfg_PVEUMin) OTE(Err_EU) ,LES(Cfg_FiltTC,0.0) OTE(Err_Filt) ];
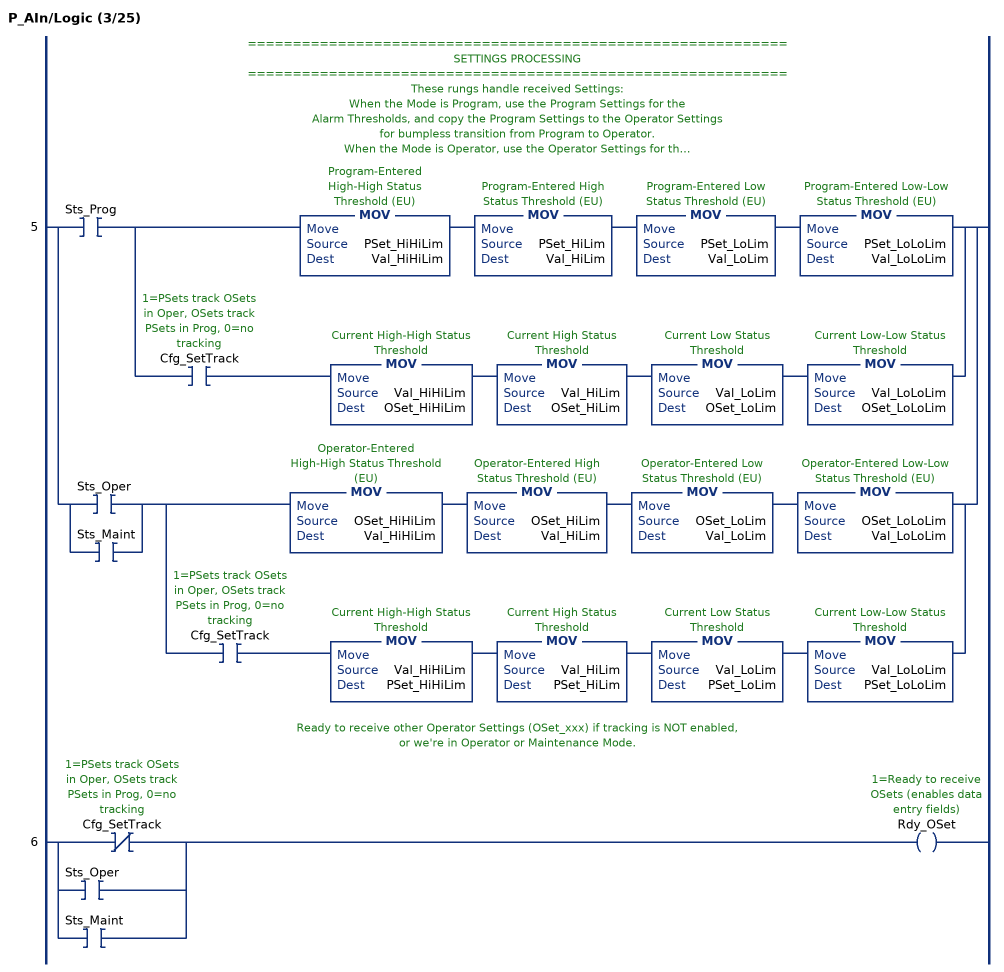
   // ============================================================
   // SETTINGS PROCESSING
   // ============================================================
   // These rungs handle received Settings:
   // When the Mode is Program, use the Program Settings for the
   // Alarm Thresholds, and copy the Program Settings to the Operator Settings
   // for bumpless transition from Program to Operator.
   // When the Mode is Operator, use the Operator Settings for the
   // Alarm Thresholds, and copy the Operator Settings to the Program Settings
   // for bumpless transition from Operator to Program.
   5: [XIC(Sts_Prog) [MOV(PSet_HiHiLim,Val_HiHiLim) MOV(PSet_HiLim,Val_HiLim) MOV(PSet_LoLim,Val_LoLim) MOV(PSet_LoLoLim,Val_LoLoLim) ,XIC(Cfg_SetTrack) MOV(Val_HiHiLim,OSet_HiHiLim) MOV(Val_HiLim,OSet_HiLim) MOV(Val_LoLim,OSet_LoLim) MOV(Val_LoLoLim,OSet_LoLoLim) ] ,[XIC(Sts_Oper) ,XIC(Sts_Maint) ] [MOV(OSet_HiHiLim,Val_HiHiLim) MOV(OSet_HiLim,Val_HiLim) MOV(OSet_LoLim,Val_LoLim) MOV(OSet_LoLoLim,Val_LoLoLim) ,XIC(Cfg_SetTrack) MOV(Val_HiHiLim,PSet_HiHiLim) MOV(Val_HiLim,PSet_HiLim) MOV(Val_LoLim,PSet_LoLim) MOV(Val_LoLoLim,PSet_LoLoLim) ] ];
   // Ready to receive other Operator Settings (OSet_xxx) if tracking is NOT enabled,
   // or we're in Operator or Maintenance Mode.
   6: [XIO(Cfg_SetTrack) ,XIC(Sts_Oper) ,XIC(Sts_Maint) ]OTE(Rdy_OSet);
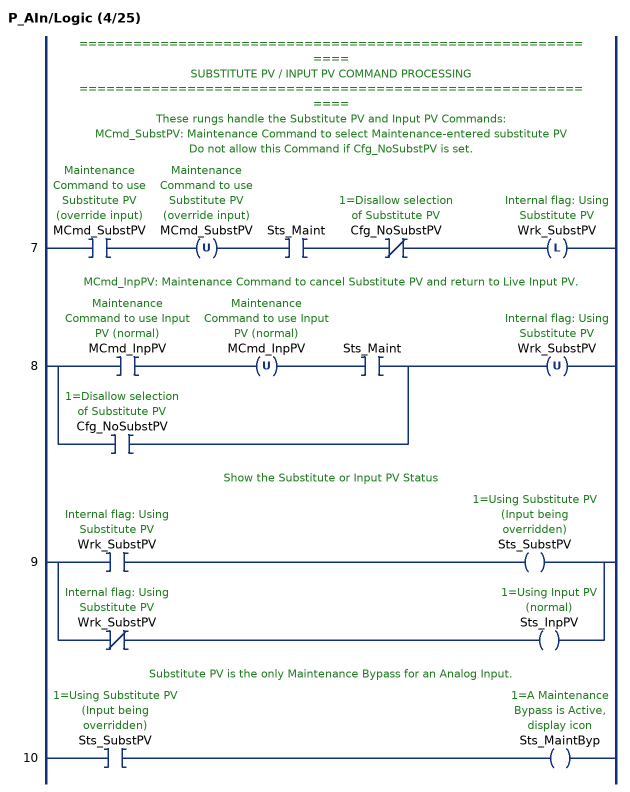
   // ============================================================
   // SUBSTITUTE PV / INPUT PV COMMAND PROCESSING
   // ============================================================
   // These rungs handle the Substitute PV and Input PV Commands:
   // MCmd_SubstPV: Maintenance Command to select Maintenance-entered substitute PV
   // Do not allow this Command if Cfg_NoSubstPV is set.
   7: XIC(MCmd_SubstPV)OTU(MCmd_SubstPV)XIC(Sts_Maint)XIO(Cfg_NoSubstPV)OTL(Wrk_SubstPV);
   // MCmd_InpPV: Maintenance Command to cancel Substitute PV and return to Live Input PV.
   8: [XIC(MCmd_InpPV) OTU(MCmd_InpPV) XIC(Sts_Maint) ,XIC(Cfg_NoSubstPV) ]OTU(Wrk_SubstPV);
   // Show the Substitute or Input PV Status
   9: [XIC(Wrk_SubstPV) OTE(Sts_SubstPV) ,XIO(Wrk_SubstPV) OTE(Sts_InpPV) ];
   // Substitute PV is the only Maintenance Bypass for an Analog Input.
   10: XIC(Sts_SubstPV)OTE(Sts_MaintByp);
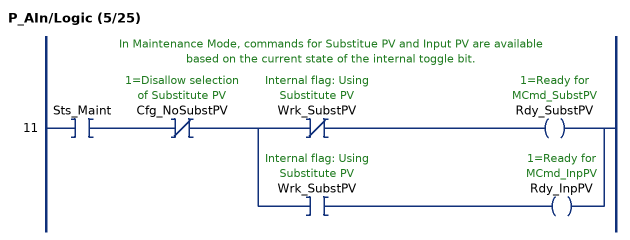
   // In Maintenance Mode, commands for Substitue PV and Input PV are available
   // based on the current state of the internal toggle bit.
   11: XIC(Sts_Maint)XIO(Cfg_NoSubstPV)[XIO(Wrk_SubstPV) OTE(Rdy_SubstPV) ,XIC(Wrk_SubstPV) OTE(Rdy_InpPV) ];
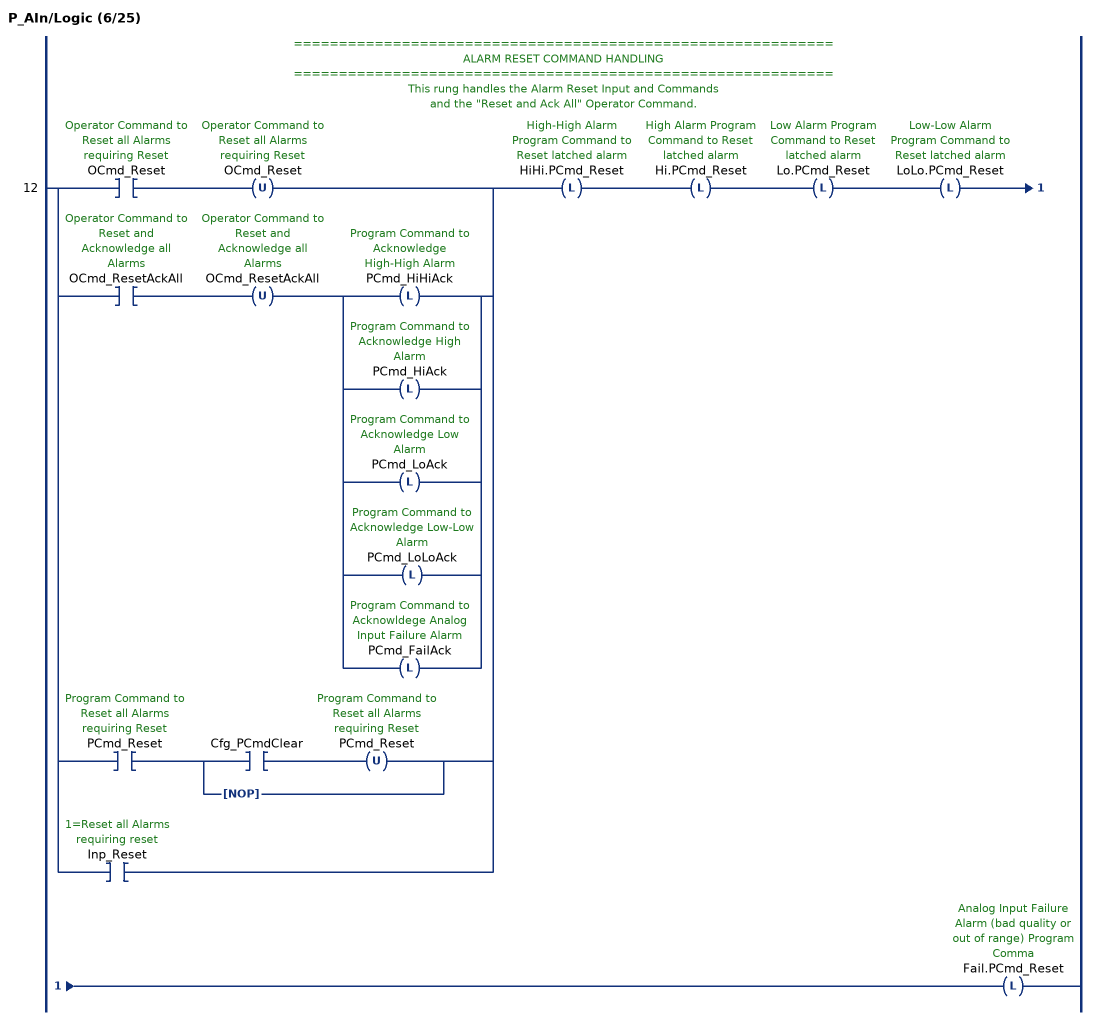
   // ============================================================
   // ALARM RESET COMMAND HANDLING
   // ============================================================
   // This rung handles the Alarm Reset Input and Commands
   // and the "Reset and Ack All" Operator Command.
   12: [XIC(OCmd_Reset) OTU(OCmd_Reset) ,XIC(OCmd_ResetAckAll) OTU(OCmd_ResetAckAll) [OTL(PCmd_HiHiAck) ,OTL(PCmd_HiAck) ,OTL(PCmd_LoAck) ,OTL(PCmd_LoLoAck) ,OTL(PCmd_FailAck) ] ,XIC(PCmd_Reset) [XIC(Cfg_PCmdClear) OTU(PCmd_Reset) ,NOP() ] ,XIC(Inp_Reset) ]OTL(HiHi.PCmd_Reset)OTL(Hi.PCmd_Reset)OTL(Lo.PCmd_Reset)OTL(LoLo.PCmd_Reset)OTL(Fail.PCmd_Reset);
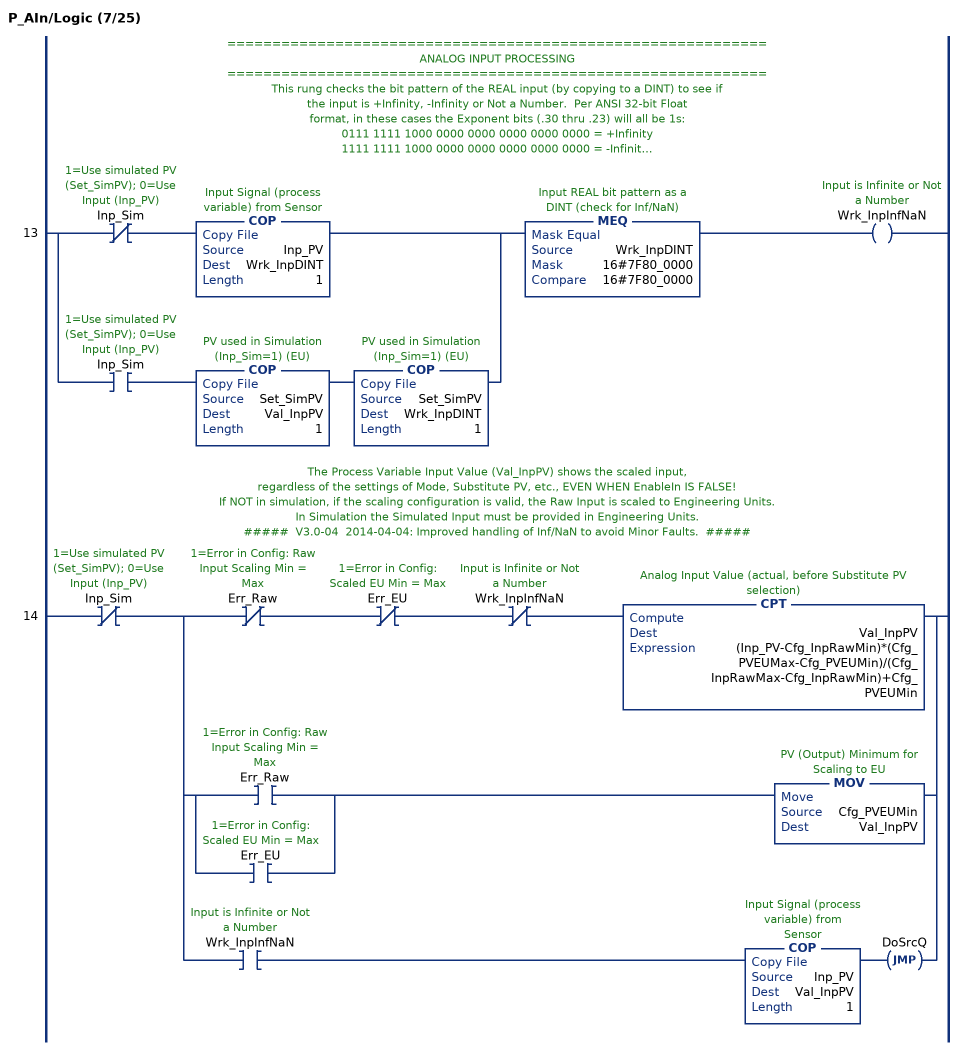
   // ============================================================
   // ANALOG INPUT PROCESSING
   // ============================================================
   // This rung checks the bit pattern of the REAL input (by copying to a DINT) to see if
   // the input is +Infinity, -Infinity or Not a Number.  Per ANSI 32-bit Float
   // format, in these cases the Exponent bits (.30 thru .23) will all be 1s:
   // 0111 1111 1000 0000 0000 0000 0000 0000 = +Infinity
   // 1111 1111 1000 0000 0000 0000 0000 0000 = -Infinity
   // x111 1111 1xxx xxxx xxxx xxxx xxxx xxxx = Not a Number
   // #####  V3.0-04  2014-04-04: Improved handling of Inf/NaN to avoid Minor Faults.  #####
   13: [XIO(Inp_Sim) COP(Inp_PV,Wrk_InpDINT,1) ,XIC(Inp_Sim) COP(Set_SimPV,Val_InpPV,1) COP(Set_SimPV,Wrk_InpDINT,1) ]MEQ(Wrk_InpDINT,16#7F80_0000,16#7F80_0000)OTE(Wrk_InpInfNaN);
   // The Process Variable Input Value (Val_InpPV) shows the scaled input,
   // regardless of the settings of Mode, Substitute PV, etc., EVEN WHEN EnableIn IS FALSE!
   // If NOT in simulation, if the scaling configuration is valid, the Raw Input is scaled to Engineering Units.
   // In Simulation the Simulated Input must be provided in Engineering Units.
   // #####  V3.0-04  2014-04-04: Improved handling of Inf/NaN to avoid Minor Faults.  #####
   14: XIO(Inp_Sim)[XIO(Err_Raw) XIO(Err_EU) XIO(Wrk_InpInfNaN) CPT(Val_InpPV,(Inp_PV-Cfg_InpRawMin)*(Cfg_PVEUMax-Cfg_PVEUMin)/(Cfg_InpRawMax-Cfg_InpRawMin)+Cfg_PVEUMin) ,[XIC(Err_Raw) ,XIC(Err_EU) ] MOV(Cfg_PVEUMin,Val_InpPV) ,XIC(Wrk_InpInfNaN) COP(Inp_PV,Val_InpPV,1) JMP(DoSrcQ) ];
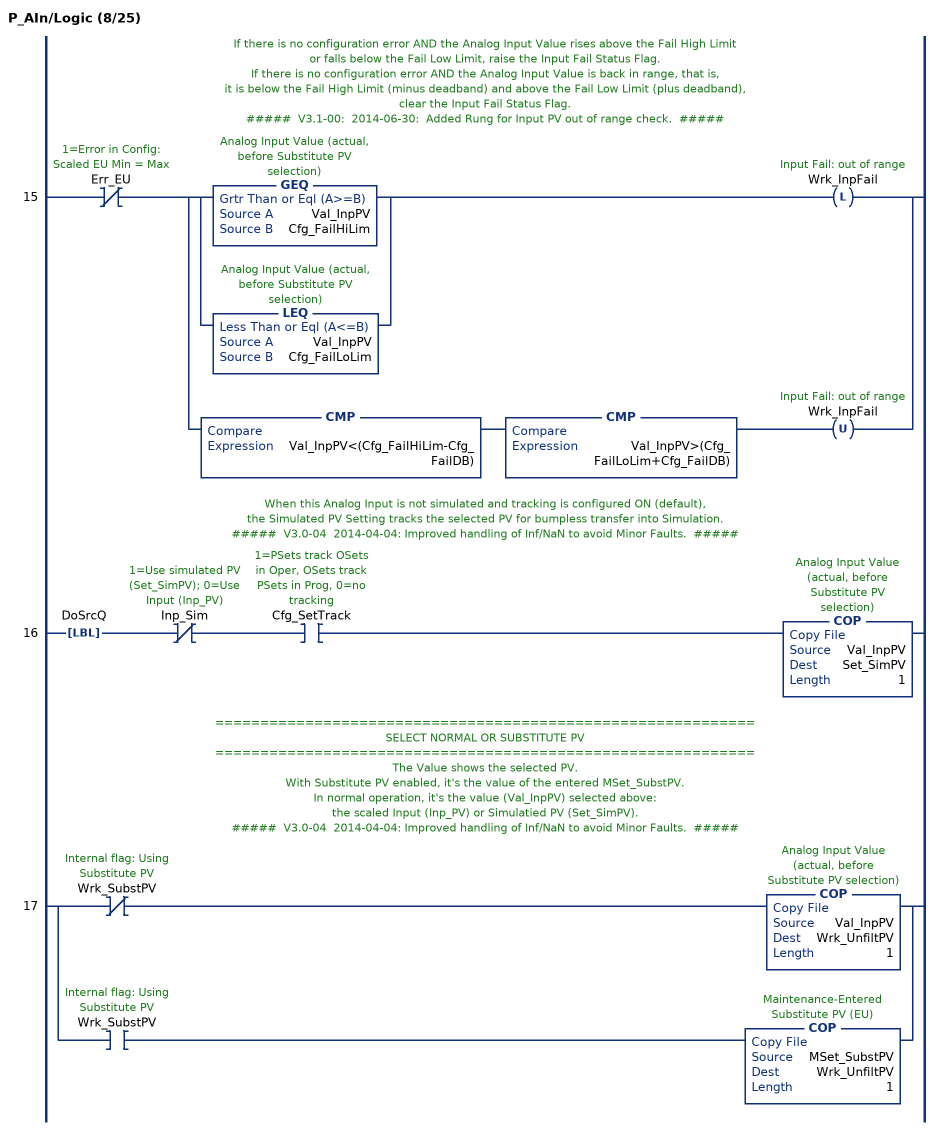
   // If there is no configuration error AND the Analog Input Value rises above the Fail High Limit
   // or falls below the Fail Low Limit, raise the Input Fail Status Flag.
   // If there is no configuration error AND the Analog Input Value is back in range, that is,
   // it is below the Fail High Limit (minus deadband) and above the Fail Low Limit (plus deadband),
   // clear the Input Fail Status Flag.
   // #####  V3.1-00:  2014-06-30:  Added Rung for Input PV out of range check.  #####
   15: XIO(Err_EU)[[GEQ(Val_InpPV,Cfg_FailHiLim) ,LEQ(Val_InpPV,Cfg_FailLoLim) ] OTL(Wrk_InpFail) ,CMP(Val_InpPV<(Cfg_FailHiLim-Cfg_FailDB)) CMP(Val_InpPV>(Cfg_FailLoLim+Cfg_FailDB)) OTU(Wrk_InpFail) ];
   // When this Analog Input is not simulated and tracking is configured ON (default),
   // the Simulated PV Setting tracks the selected PV for bumpless transfer into Simulation.
   // #####  V3.0-04  2014-04-04: Improved handling of Inf/NaN to avoid Minor Faults.  #####
   16: LBL(DoSrcQ)XIO(Inp_Sim)XIC(Cfg_SetTrack)COP(Val_InpPV,Set_SimPV,1);
   // ============================================================
   // SELECT NORMAL OR SUBSTITUTE PV
   // ============================================================
   // The Value shows the selected PV.
   // With Substitute PV enabled, it's the value of the entered MSet_SubstPV.
   // In normal operation, it's the value (Val_InpPV) selected above:
   // the scaled Input (Inp_PV) or Simulatied PV (Set_SimPV).
   // #####  V3.0-04  2014-04-04: Improved handling of Inf/NaN to avoid Minor Faults.  #####
   17: [XIO(Wrk_SubstPV) COP(Val_InpPV,Wrk_UnfiltPV,1) ,XIC(Wrk_SubstPV) COP(MSet_SubstPV,Wrk_UnfiltPV,1) ];
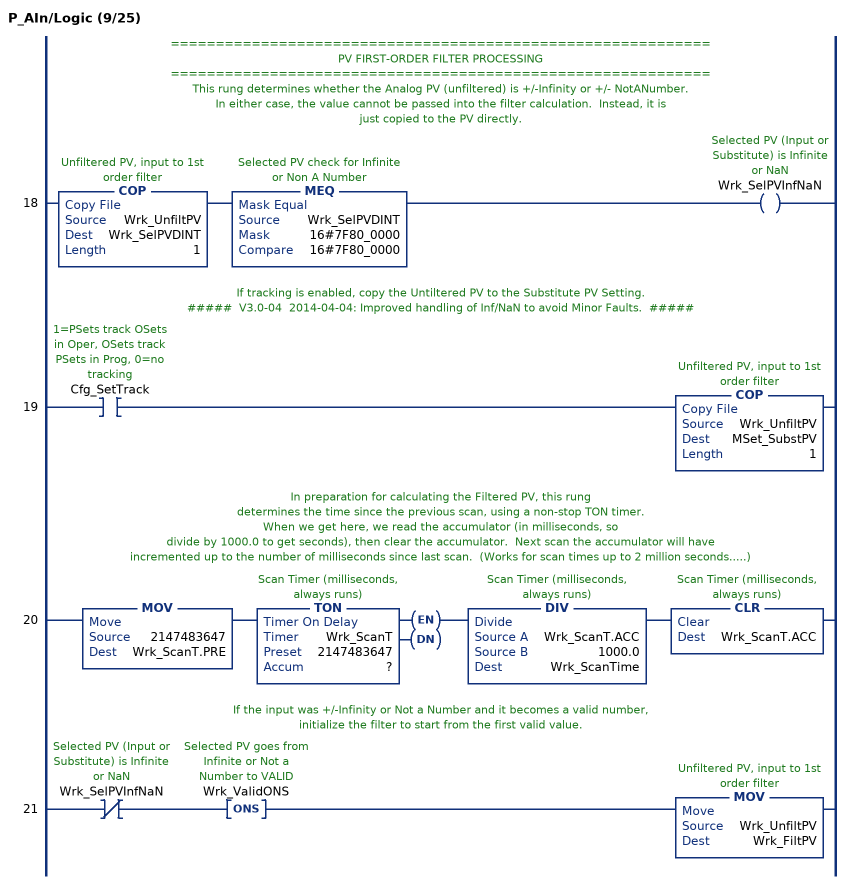
   // ============================================================
   // PV FIRST-ORDER FILTER PROCESSING
   // ============================================================
   // This rung determines whether the Analog PV (unfiltered) is +/-Infinity or +/- NotANumber.
   // In either case, the value cannot be passed into the filter calculation.  Instead, it is
   // just copied to the PV directly.
   18: COP(Wrk_UnfiltPV,Wrk_SelPVDINT,1)MEQ(Wrk_SelPVDINT,16#7F80_0000,16#7F80_0000)OTE(Wrk_SelPVInfNaN);
   // If tracking is enabled, copy the Untiltered PV to the Substitute PV Setting.
   // #####  V3.0-04  2014-04-04: Improved handling of Inf/NaN to avoid Minor Faults.  #####
   19: XIC(Cfg_SetTrack)COP(Wrk_UnfiltPV,MSet_SubstPV,1);
   // In preparation for calculating the Filtered PV, this rung
   // determines the time since the previous scan, using a non-stop TON timer.
   // When we get here, we read the accumulator (in milliseconds, so
   // divide by 1000.0 to get seconds), then clear the accumulator.  Next scan the accumulator will have
   // incremented up to the number of milliseconds since last scan.  (Works for scan times up to 2 million seconds.....)
   20: MOV(2147483647,Wrk_ScanT.PRE)TON(Wrk_ScanT,?,?)DIV(Wrk_ScanT.ACC,1000.0,Wrk_ScanTime)CLR(Wrk_ScanT.ACC);
   // If the input was +/-Infinity or Not a Number and it becomes a valid number,
   // initialize the filter to start from the first valid value.
   21: XIO(Wrk_SelPVInfNaN)ONS(Wrk_ValidONS)MOV(Wrk_UnfiltPV,Wrk_FiltPV);
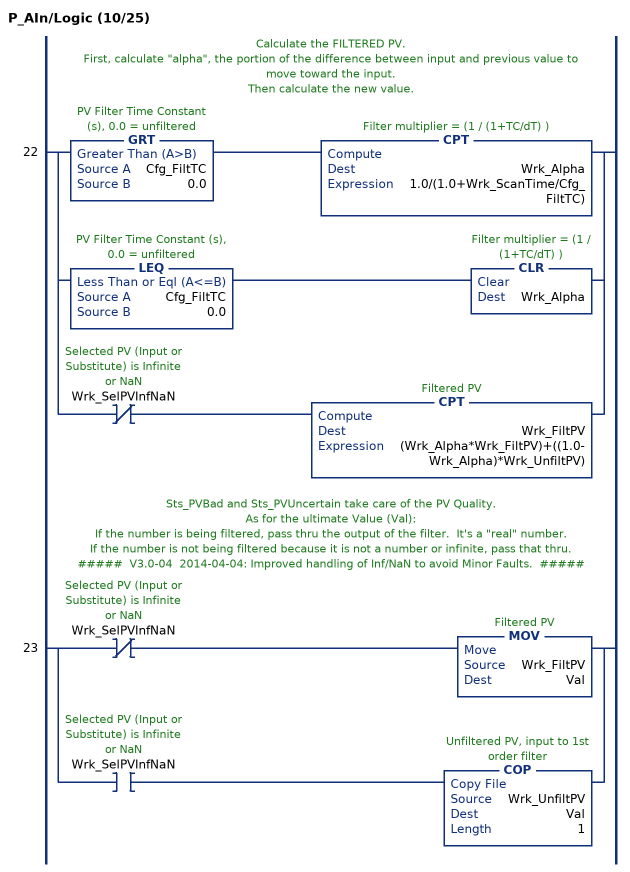
   // Calculate the FILTERED PV.
   // First, calculate "alpha", the portion of the difference between input and previous value to move toward the input.
   // Then calculate the new value.
   22: [GRT(Cfg_FiltTC,0.0) CPT(Wrk_Alpha,1.0/(1.0+Wrk_ScanTime/Cfg_FiltTC)) ,LEQ(Cfg_FiltTC,0.0) CLR(Wrk_Alpha) ,XIO(Wrk_SelPVInfNaN) CPT(Wrk_FiltPV,(Wrk_Alpha*Wrk_FiltPV)+((1.0-Wrk_Alpha)*Wrk_UnfiltPV)) ];
   // Sts_PVBad and Sts_PVUncertain take care of the PV Quality.
   // As for the ultimate Value (Val):
   // If the number is being filtered, pass thru the output of the filter.  It's a "real" number.
   // If the number is not being filtered because it is not a number or infinite, pass that thru.
   // #####  V3.0-04  2014-04-04: Improved handling of Inf/NaN to avoid Minor Faults.  #####
   23: [XIO(Wrk_SelPVInfNaN) MOV(Wrk_FiltPV,Val) ,XIC(Wrk_SelPVInfNaN) COP(Wrk_UnfiltPV,Val,1) ];
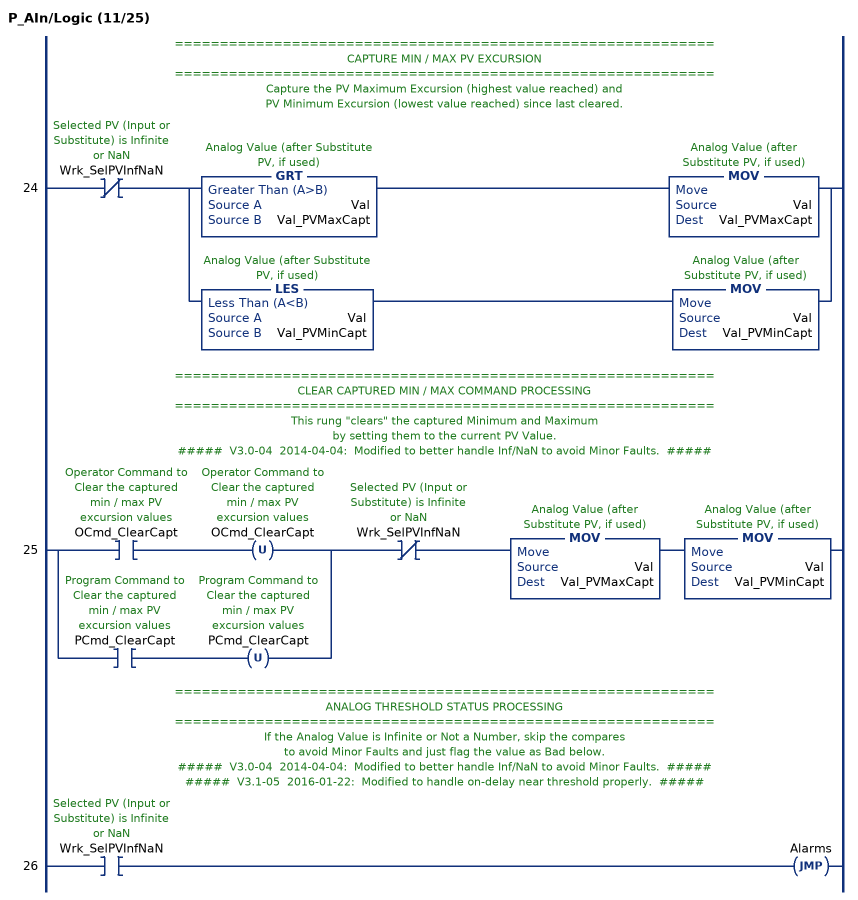
   // ============================================================
   // CAPTURE MIN / MAX PV EXCURSION
   // ============================================================
   // Capture the PV Maximum Excursion (highest value reached) and
   // PV Minimum Excursion (lowest value reached) since last cleared.
   24: XIO(Wrk_SelPVInfNaN)[GRT(Val,Val_PVMaxCapt) MOV(Val,Val_PVMaxCapt) ,LES(Val,Val_PVMinCapt) MOV(Val,Val_PVMinCapt) ];
   // ============================================================
   // CLEAR CAPTURED MIN / MAX COMMAND PROCESSING
   // ============================================================
   // This rung "clears" the captured Minimum and Maximum
   // by setting them to the current PV Value.
   // #####  V3.0-04  2014-04-04:  Modified to better handle Inf/NaN to avoid Minor Faults.  #####
   25: [XIC(OCmd_ClearCapt) OTU(OCmd_ClearCapt) ,XIC(PCmd_ClearCapt) OTU(PCmd_ClearCapt) ]XIO(Wrk_SelPVInfNaN)MOV(Val,Val_PVMaxCapt)MOV(Val,Val_PVMinCapt);
   // ============================================================
   // ANALOG THRESHOLD STATUS PROCESSING
   // ============================================================
   // If the Analog Value is Infinite or Not a Number, skip the compares
   // to avoid Minor Faults and just flag the value as Bad below.
   // #####  V3.0-04  2014-04-04:  Modified to better handle Inf/NaN to avoid Minor Faults.  #####
   // #####  V3.1-05  2016-01-22:  Modified to handle on-delay near threshold properly.  #####
   26: XIC(Wrk_SelPVInfNaN)JMP(Alarms);
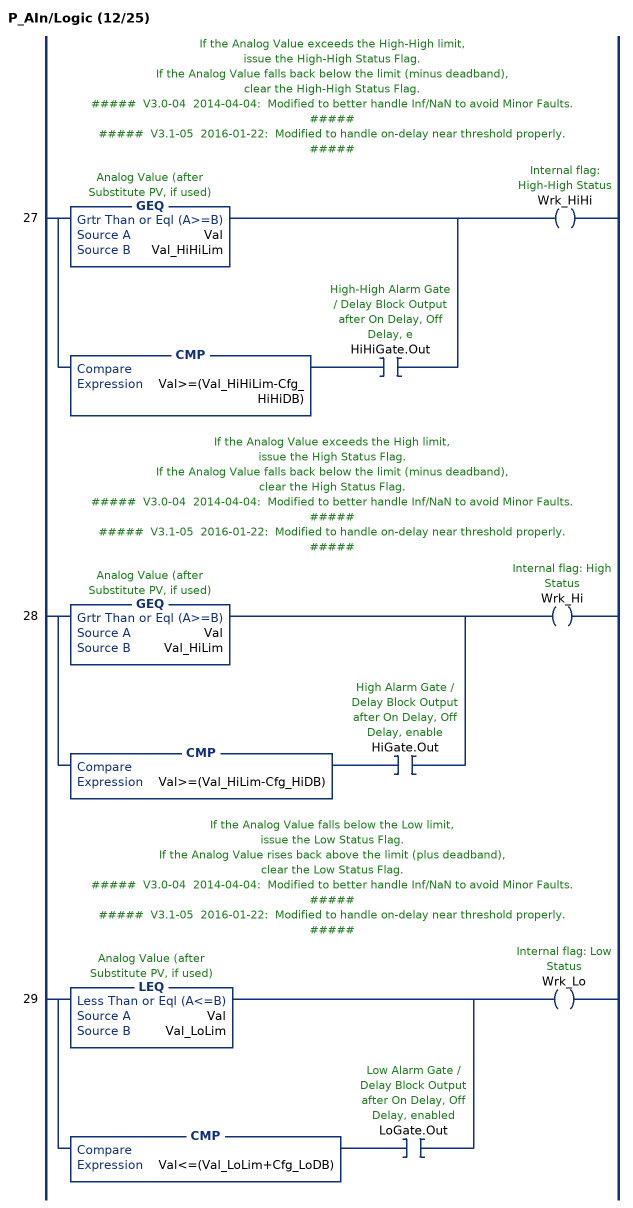
   // If the Analog Value exceeds the High-High limit,
   // issue the High-High Status Flag.
   // If the Analog Value falls back below the limit (minus deadband),
   // clear the High-High Status Flag.
   // #####  V3.0-04  2014-04-04:  Modified to better handle Inf/NaN to avoid Minor Faults.  #####
   // #####  V3.1-05  2016-01-22:  Modified to handle on-delay near threshold properly.  #####
   27: [GEQ(Val,Val_HiHiLim) ,CMP(Val>=(Val_HiHiLim-Cfg_HiHiDB)) XIC(HiHiGate.Out) ]OTE(Wrk_HiHi);
   // If the Analog Value exceeds the High limit,
   // issue the High Status Flag.
   // If the Analog Value falls back below the limit (minus deadband),
   // clear the High Status Flag.
   // #####  V3.0-04  2014-04-04:  Modified to better handle Inf/NaN to avoid Minor Faults.  #####
   // #####  V3.1-05  2016-01-22:  Modified to handle on-delay near threshold properly.  #####
   28: [GEQ(Val,Val_HiLim) ,CMP(Val>=(Val_HiLim-Cfg_HiDB)) XIC(HiGate.Out) ]OTE(Wrk_Hi);
   // If the Analog Value falls below the Low limit,
   // issue the Low Status Flag.
   // If the Analog Value rises back above the limit (plus deadband),
   // clear the Low Status Flag.
   // #####  V3.0-04  2014-04-04:  Modified to better handle Inf/NaN to avoid Minor Faults.  #####
   // #####  V3.1-05  2016-01-22:  Modified to handle on-delay near threshold properly.  #####
   29: [LEQ(Val,Val_LoLim) ,CMP(Val<=(Val_LoLim+Cfg_LoDB)) XIC(LoGate.Out) ]OTE(Wrk_Lo);
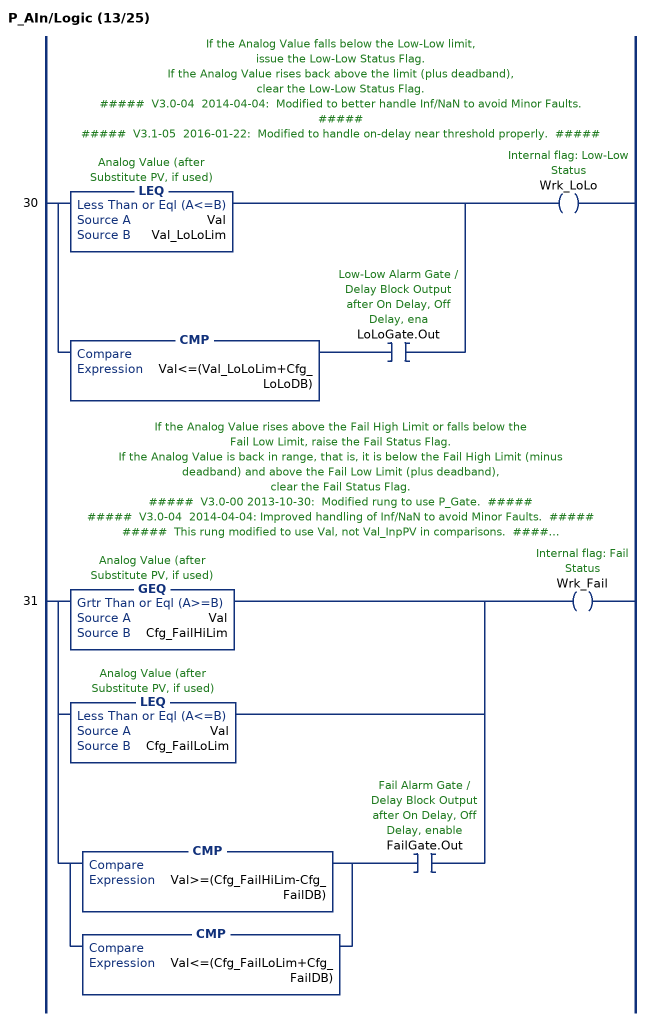
   // If the Analog Value falls below the Low-Low limit,
   // issue the Low-Low Status Flag.
   // If the Analog Value rises back above the limit (plus deadband),
   // clear the Low-Low Status Flag.
   // #####  V3.0-04  2014-04-04:  Modified to better handle Inf/NaN to avoid Minor Faults.  #####
   // #####  V3.1-05  2016-01-22:  Modified to handle on-delay near threshold properly.  #####
   30: [LEQ(Val,Val_LoLoLim) ,CMP(Val<=(Val_LoLoLim+Cfg_LoLoDB)) XIC(LoLoGate.Out) ]OTE(Wrk_LoLo);
   // If the Analog Value rises above the Fail High Limit or falls below the
   // Fail Low Limit, raise the Fail Status Flag.
   // If the Analog Value is back in range, that is, it is below the Fail High Limit (minus
   // deadband) and above the Fail Low Limit (plus deadband),
   // clear the Fail Status Flag.
   // #####  V3.0-00 2013-10-30:  Modified rung to use P_Gate.  #####
   // #####  V3.0-04  2014-04-04: Improved handling of Inf/NaN to avoid Minor Faults.  #####
   // #####  This rung modified to use Val, not Val_InpPV in comparisons.  #####
   // #####  V3.1-05  2016-01-22:  Modified to handle on-delay near threshold properly.  #####
   31: [[GEQ(Val,Cfg_FailHiLim) ,LEQ(Val,Cfg_FailLoLim) ] ,[CMP(Val>=(Cfg_FailHiLim-Cfg_FailDB)) ,CMP(Val<=(Cfg_FailLoLim+Cfg_FailDB)) ] XIC(FailGate.Out) ]OTE(Wrk_Fail);
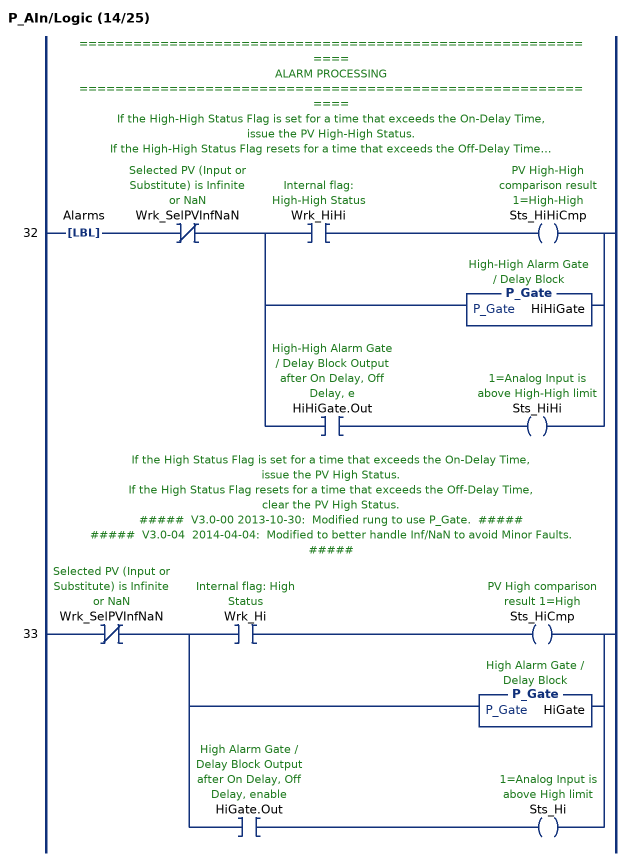
   // ============================================================
   // ALARM PROCESSING
   // ============================================================
   // If the High-High Status Flag is set for a time that exceeds the On-Delay Time,
   // issue the PV High-High Status.
   // If the High-High Status Flag resets for a time that exceeds the Off-Delay Time,
   // clear the PV High-High Status.
   // #####  V3.0-00 2013-10-30:  Modified rung to use P_Gate.  #####
   // #####  V3.0-04  2014-04-04:  Modified to better handle Inf/NaN to avoid Minor Faults.  #####
   32: LBL(Alarms)XIO(Wrk_SelPVInfNaN)[XIC(Wrk_HiHi) OTE(Sts_HiHiCmp) ,P_Gate(HiHiGate) ,XIC(HiHiGate.Out) OTE(Sts_HiHi) ];
   // If the High Status Flag is set for a time that exceeds the On-Delay Time,
   // issue the PV High Status.
   // If the High Status Flag resets for a time that exceeds the Off-Delay Time,
   // clear the PV High Status.
   // #####  V3.0-00 2013-10-30:  Modified rung to use P_Gate.  #####
   // #####  V3.0-04  2014-04-04:  Modified to better handle Inf/NaN to avoid Minor Faults.  #####
   33: XIO(Wrk_SelPVInfNaN)[XIC(Wrk_Hi) OTE(Sts_HiCmp) ,P_Gate(HiGate) ,XIC(HiGate.Out) OTE(Sts_Hi) ];
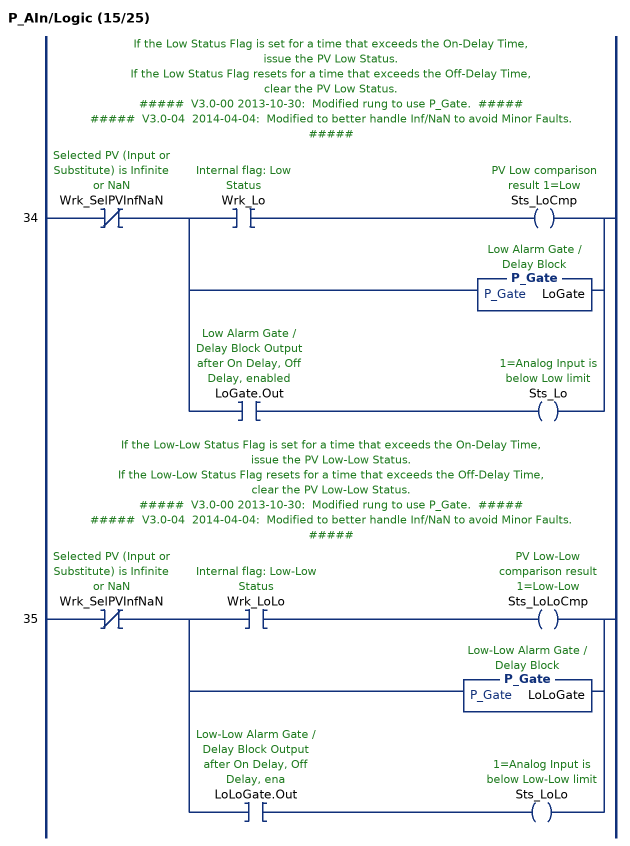
   // If the Low Status Flag is set for a time that exceeds the On-Delay Time,
   // issue the PV Low Status.
   // If the Low Status Flag resets for a time that exceeds the Off-Delay Time,
   // clear the PV Low Status.
   // #####  V3.0-00 2013-10-30:  Modified rung to use P_Gate.  #####
   // #####  V3.0-04  2014-04-04:  Modified to better handle Inf/NaN to avoid Minor Faults.  #####
   34: XIO(Wrk_SelPVInfNaN)[XIC(Wrk_Lo) OTE(Sts_LoCmp) ,P_Gate(LoGate) ,XIC(LoGate.Out) OTE(Sts_Lo) ];
   // If the Low-Low Status Flag is set for a time that exceeds the On-Delay Time,
   // issue the PV Low-Low Status.
   // If the Low-Low Status Flag resets for a time that exceeds the Off-Delay Time,
   // clear the PV Low-Low Status.
   // #####  V3.0-00 2013-10-30:  Modified rung to use P_Gate.  #####
   // #####  V3.0-04  2014-04-04:  Modified to better handle Inf/NaN to avoid Minor Faults.  #####
   35: XIO(Wrk_SelPVInfNaN)[XIC(Wrk_LoLo) OTE(Sts_LoLoCmp) ,P_Gate(LoLoGate) ,XIC(LoLoGate.Out) OTE(Sts_LoLo) ];
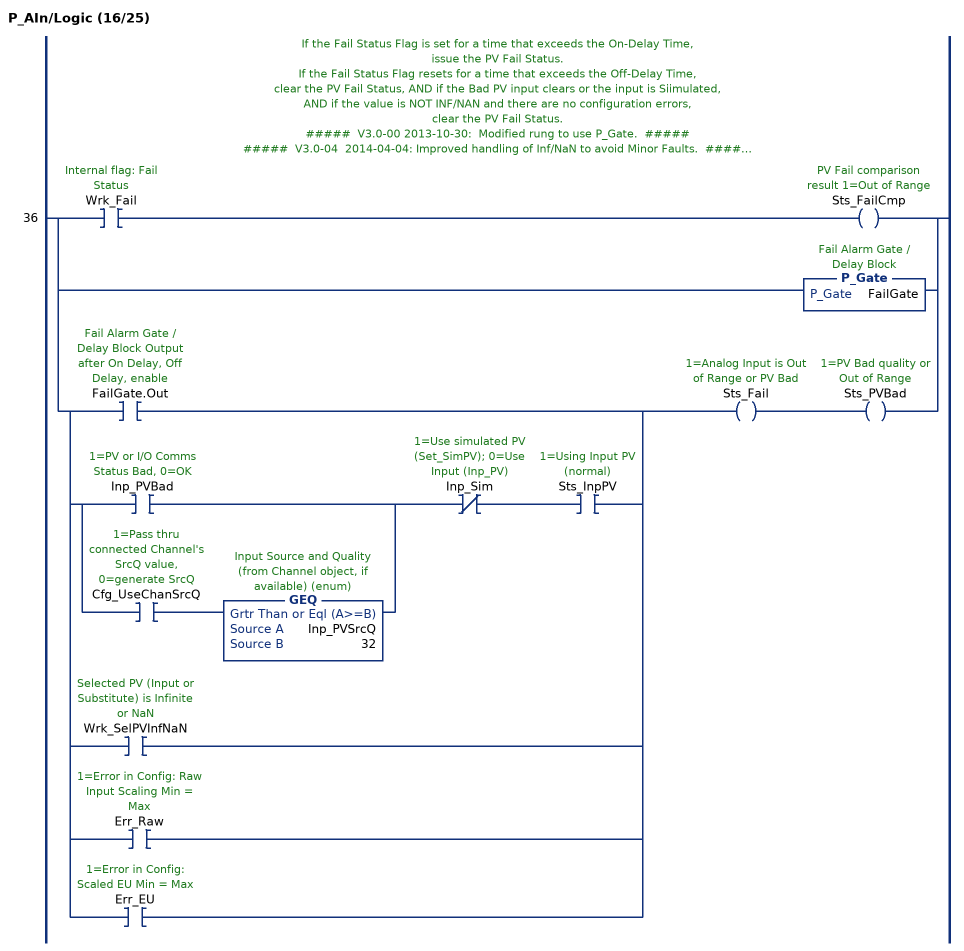
   // If the Fail Status Flag is set for a time that exceeds the On-Delay Time,
   // issue the PV Fail Status.
   // If the Fail Status Flag resets for a time that exceeds the Off-Delay Time,
   // clear the PV Fail Status, AND if the Bad PV input clears or the input is Siimulated,
   // AND if the value is NOT INF/NAN and there are no configuration errors,
   // clear the PV Fail Status.
   // #####  V3.0-00 2013-10-30:  Modified rung to use P_Gate.  #####
   // #####  V3.0-04  2014-04-04: Improved handling of Inf/NaN to avoid Minor Faults.  #####
   // #####  V3.1-00  2014-06-30:  Modified to use input channel Source/Quality enumeration.  #####
   // #####  V3.5-02  2016-03-28:  Modified to add Cfg_UseChanSrcQ.  #####
   36: [XIC(Wrk_Fail) OTE(Sts_FailCmp) ,P_Gate(FailGate) ,[XIC(FailGate.Out) ,[XIC(Inp_PVBad) ,XIC(Cfg_UseChanSrcQ) GEQ(Inp_PVSrcQ,32) ] XIO(Inp_Sim) XIC(Sts_InpPV) ,XIC(Wrk_SelPVInfNaN) ,XIC(Err_Raw) ,XIC(Err_EU) ] OTE(Sts_Fail) OTE(Sts_PVBad) ];
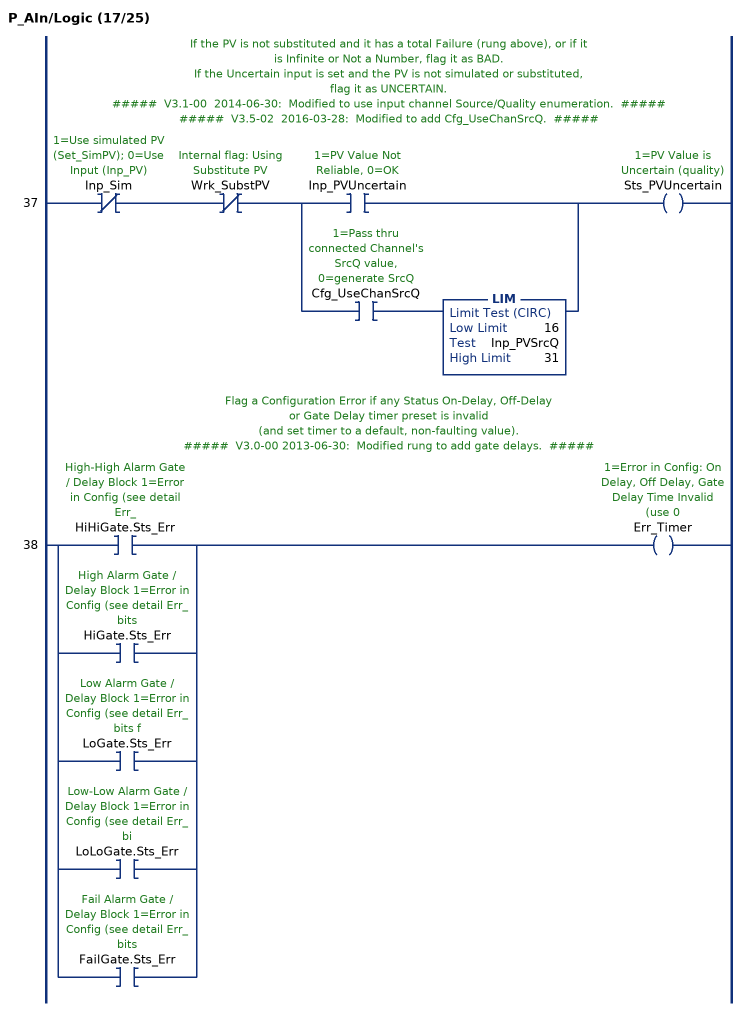
   // If the PV is not substituted and it has a total Failure (rung above), or if it
   // is Infinite or Not a Number, flag it as BAD.
   // If the Uncertain input is set and the PV is not simulated or substituted,
   // flag it as UNCERTAIN.
   // #####  V3.1-00  2014-06-30:  Modified to use input channel Source/Quality enumeration.  #####
   // #####  V3.5-02  2016-03-28:  Modified to add Cfg_UseChanSrcQ.  #####
   37: XIO(Inp_Sim)XIO(Wrk_SubstPV)[XIC(Inp_PVUncertain) ,XIC(Cfg_UseChanSrcQ) LIM(16,Inp_PVSrcQ,31) ]OTE(Sts_PVUncertain);
   // Flag a Configuration Error if any Status On-Delay, Off-Delay
   // or Gate Delay timer preset is invalid
   // (and set timer to a default, non-faulting value).
   // #####  V3.0-00 2013-06-30:  Modified rung to add gate delays.  #####
   38: [XIC(HiHiGate.Sts_Err) ,XIC(HiGate.Sts_Err) ,XIC(LoGate.Sts_Err) ,XIC(LoLoGate.Sts_Err) ,XIC(FailGate.Sts_Err) ]OTE(Err_Timer);
